C07376=1109.585,-100.826,-47.204,179.816,4.533,148.808
C07377=1109.580,-100.611,-47.213,179.815,4.537,148.809
C07378=1109.575,-100.396,-47.221,179.814,4.541,148.810
C07379=1109.571,-100.182,-47.230,179.814,4.545,148.811
C07380=1109.566,-99.966,-47.239,179.814,4.550,148.812
C07381=1109.561,-99.752,-47.247,179.814,4.555,148.813
C07382=1109.557,-99.538,-47.256,179.813,4.559,148.814
C07383=1109.553,-99.322,-47.264,179.813,4.562,148.815
C07384=1109.547,-99.073,-47.275,179.813,4.568,148.816
C07385=1109.542,-98.823,-47.285,179.813,4.573,148.817
C07386=1109.537,-98.574,-47.294,179.812,4.578,148.818
C07387=1109.532,-98.323,-47.304,179.812,4.582,148.820
C07388=1109.526,-98.074,-47.315,179.811,4.587,148.821
C07389=1109.520,-97.824,-47.325,179.811,4.593,148.822
C07390=1109.516,-97.575,-47.334,179.810,4.597,148.823
C07391=1109.511,-97.325,-47.345,179.810,4.602,148.824
C07392=1109.505,-97.075,-47.355,179.810,4.607,148.826
C07393=1109.499,-96.826,-47.365,179.810,4.612,148.827
C07394=1109.495,-96.576,-47.375,179.809,4.617,148.828
C07395=1109.489,-96.325,-47.385,179.809,4.622,148.829
C07396=1109.484,-96.076,-47.395,179.809,4.627,148.830
C07397=1109.479,-95.826,-47.406,179.808,4.631,148.832
C07398=1109.474,-95.576,-47.415,179.808,4.637,148.833
C07399=1109.468,-95.327,-47.425,179.807,4.642,148.834
C07400=1109.463,-95.077,-47.436,179.807,4.647,148.835
C07401=1109.458,-94.827,-47.446,179.806,4.651,148.836
C07402=1109.452,-94.578,-47.456,179.806,4.656,148.838
C07403=1109.447,-94.328,-47.466,179.806,4.661,148.839
C07404=1109.442,-94.078,-47.477,179.805,4.666,148.840
C07405=1109.437,-93.829,-47.487,179.805,4.671,148.841
C07406=1109.431,-93.579,-47.497,179.804,4.675,148.842
C07407=1109.426,-93.329,-47.508,179.804,4.680,148.844
C07408=1109.420,-93.079,-47.518,179.804,4.686,148.845
C07409=1109.416,-92.830,-47.527,179.803,4.690,148.846
C07410=1109.411,-92.580,-47.538,179.803,4.695,148.847
C07411=1109.405,-92.330,-47.548,179.803,4.700,148.848
C07412=1109.400,-92.080,-47.559,179.801,4.705,148.850
C07413=1109.394,-91.830,-47.569,179.801,4.710,148.851
C07414=1109.389,-91.581,-47.579,179.800,4.714,148.852
C07415=1109.384,-91.331,-47.589,179.800,4.720,148.853
C07416=1109.379,-91.081,-47.599,179.800,4.725,148.854
C07417=1109.373,-90.832,-47.610,179.799,4.729,148.856
C07418=1109.368,-90.582,-47.620,179.799,4.734,148.857
C07419=1109.363,-90.332,-47.630,179.799,4.739,148.858
C07420=1109.358,-90.082,-47.641,179.799,4.745,148.859
C07421=1109.352,-89.832,-47.651,179.797,4.749,148.861
C07422=1109.346,-89.583,-47.661,179.797,4.754,148.862
C07423=1109.342,-89.333,-47.673,179.797,4.760,148.863
C07424=1109.337,-89.084,-47.682,179.796,4.764,148.864
C07425=1109.332,-88.834,-47.693,179.796,4.769,148.865
C07426=1109.326,-88.584,-47.703,179.796,4.774,148.867
C07427=1109.321,-88.335,-47.713,179.796,4.779,148.868
C07428=1109.316,-88.084,-47.724,179.795,4.784,148.869
C07429=1109.310,-87.835,-47.734,179.794,4.789,148.870
C07430=1109.305,-87.585,-47.745,179.794,4.794,148.872
C07431=1109.300,-87.336,-47.756,179.794,4.799,148.873
C07432=1109.296,-87.120,-47.764,179.793,4.803,148.874
C07433=1109.291,-86.906,-47.773,179.793,4.808,148.875
C07434=1109.286,-86.692,-47.782,179.792,4.812,148.876
C07435=1109.282,-86.476,-47.791,179.793,4.817,148.877
C07436=1109.277,-86.262,-47.800,179.792,4.821,148.878
C07437=1109.273,-86.047,-47.810,179.792,4.825,148.879
C07438=1109.268,-85.832,-47.818,179.791,4.830,148.880
C07439=1109.263,-85.618,-47.827,179.791,4.834,148.881
C07440=1109.259,-85.368,-47.838,179.791,4.839,148.882
C07441=1109.253,-85.119,-47.849,179.791,4.844,148.883
C07442=1109.248,-84.868,-47.859,179.790,4.849,148.885
C07443=1109.242,-84.619,-47.869,179.790,4.854,148.886
C07444=1109.238,-84.369,-47.881,179.789,4.859,148.887
C07445=1109.232,-84.120,-47.891,179.789,4.864,148.888
C07446=1109.227,-83.869,-47.901,179.789,4.869,148.889
C07447=1109.221,-83.620,-47.912,179.789,4.875,148.891
C07448=1109.217,-83.370,-47.923,179.789,4.880,148.892
C07449=1109.211,-83.121,-47.933,179.788,4.884,148.893
C07450=1109.206,-82.870,-47.944,179.788,4.889,148.894
C07451=1109.201,-82.621,-47.955,179.787,4.894,148.895
C07452=1109.196,-82.371,-47.965,179.787,4.900,148.897
C07453=1109.190,-82.122,-47.975,179.787,4.905,148.898
C07454=1109.186,-81.872,-47.987,179.786,4.910,148.899
C07455=1109.180,-81.622,-47.997,179.786,4.915,148.900
C07456=1109.175,-81.372,-48.007,179.786,4.921,148.902
C07457=1109.170,-81.123,-48.018,179.786,4.926,148.903
C07458=1109.164,-80.873,-48.030,179.786,4.931,148.904
C07459=1109.158,-80.623,-48.040,179.786,4.936,148.905
C07460=1109.154,-80.374,-48.051,179.785,4.940,148.906
C07461=1109.148,-80.124,-48.061,179.785,4.945,148.907
C07462=1109.143,-79.874,-48.072,179.785,4.951,148.909
C07463=1109.138,-79.625,-48.083,179.784,4.956,148.910
C07464=1109.133,-79.375,-48.093,179.784,4.961,148.911
C07465=1109.128,-79.125,-48.105,179.784,4.966,148.912
C07466=1109.122,-78.875,-48.115,179.784,4.971,148.913
C07467=1109.117,-78.626,-48.127,179.784,4.976,148.914
C07468=1109.111,-78.376,-48.137,179.784,4.981,148.916
C07469=1109.106,-78.126,-48.148,179.783,4.987,148.917
C07470=1109.101,-77.877,-48.158,179.783,4.992,148.918
C07471=1109.096,-77.627,-48.169,179.783,4.997,148.919
C07472=1109.090,-77.377,-48.181,179.782,5.002,148.921
C07473=1109.085,-77.127,-48.191,179.782,5.008,148.922
C07474=1109.080,-76.877,-48.202,179.782,5.013,148.923
C07475=1109.075,-76.628,-48.213,179.782,5.018,148.924
C07476=1109.070,-76.378,-48.224,179.782,5.023,148.925
C07477=1109.064,-76.128,-48.235,179.782,5.028,148.926
C07478=1109.059,-75.879,-48.246,179.782,5.033,148.928
C07479=1109.054,-75.629,-48.257,179.782,5.038,148.929
C07480=1109.049,-75.380,-48.268,179.782,5.043,148.930
C07481=1109.044,-75.129,-48.278,179.782,5.048,148.931
C07482=1109.038,-74.880,-48.290,179.781,5.053,148.932
C07483=1109.033,-74.631,-48.301,179.781,5.059,148.933
C07484=1109.028,-74.380,-48.311,179.781,5.064,148.934
C07485=1109.023,-74.131,-48.322,179.781,5.069,148.936
C07486=1109.017,-73.881,-48.334,179.781,5.074,148.937
C07487=1109.012,-73.631,-48.345,179.781,5.080,148.938
C07488=1109.008,-73.417,-48.354,179.781,5.084,148.939
C07489=1109.003,-73.202,-48.364,179.781,5.089,148.940
C07490=1108.999,-72.988,-48.373,179.781,5.093,148.941
C07491=1108.994,-72.773,-48.383,179.781,5.098,148.942
C07492=1108.989,-72.559,-48.392,179.781,5.102,148.943
C07493=1108.985,-72.343,-48.402,179.781,5.106,148.944
C07494=1108.981,-72.129,-48.411,179.781,5.110,148.945
C07495=1108.976,-71.914,-48.421,179.781,5.115,148.946
C07496=1108.972,-71.665,-48.432,179.781,5.120,148.947
C07497=1108.965,-71.415,-48.443,179.781,5.125,148.948
C07498=1108.960,-71.165,-48.454,179.781,5.131,148.949
C07499=1108.956,-70.916,-48.465,179.781,5.136,148.950
C07500=1108.949,-70.666,-48.476,179.781,5.141,148.951
C07501=1108.945,-70.416,-48.488,179.781,5.146,148.952
C07502=1108.940,-70.167,-48.499,179.781,5.151,148.954
C07503=1108.935,-69.917,-48.511,179.781,5.156,148.955
C07504=1108.929,-69.667,-48.521,179.781,5.161,148.956
C07505=1108.924,-69.418,-48.532,179.781,5.166,148.957
C07506=1108.919,-69.168,-48.544,179.781,5.172,148.958
C07507=1108.914,-68.919,-48.555,179.781,5.177,148.959
C07508=1108.908,-68.668,-48.566,179.781,5.182,148.960
C07509=1108.903,-68.418,-48.578,179.782,5.187,148.961
C07510=1108.899,-68.169,-48.589,179.781,5.192,148.962
C07511=1108.892,-67.920,-48.600,179.781,5.197,148.964
C07512=1108.888,-67.670,-48.612,179.782,5.202,148.964
C07513=1108.882,-67.420,-48.624,179.782,5.207,148.966
C07514=1108.877,-67.170,-48.634,179.781,5.212,148.967
C07515=1108.871,-66.921,-48.646,179.782,5.218,148.968
C07516=1108.867,-66.671,-48.657,179.782,5.223,148.969
C07517=1108.862,-66.421,-48.668,179.782,5.228,148.970
C07518=1108.857,-66.171,-48.680,179.783,5.233,148.971
C07519=1108.851,-65.922,-48.691,179.782,5.238,148.972
C07520=1108.846,-65.673,-48.703,179.783,5.243,148.973
C07521=1108.841,-65.422,-48.713,179.783,5.248,148.974
C07522=1108.835,-65.172,-48.725,179.783,5.252,148.975
C07523=1108.831,-64.923,-48.737,179.784,5.258,148.976
C07524=1108.825,-64.674,-48.748,179.783,5.264,148.977
C07525=1108.820,-64.424,-48.759,179.784,5.268,148.978
C07526=1108.815,-64.174,-48.771,179.784,5.273,148.980
C07527=1108.810,-63.924,-48.783,179.784,5.278,148.981
C07528=1108.804,-63.674,-48.794,179.784,5.283,148.981
C07529=1108.799,-63.425,-48.805,179.784,5.288,148.983
C07530=1108.794,-63.176,-48.817,179.785,5.294,148.984
C07531=1108.789,-62.926,-48.829,179.785,5.299,148.985
C07532=1108.784,-62.676,-48.840,179.786,5.304,148.986
C07533=1108.779,-62.426,-48.852,179.786,5.309,148.987
C07534=1108.773,-62.176,-48.864,179.786,5.313,148.988
C07535=1108.767,-61.927,-48.875,179.786,5.318,148.989
C07536=1108.763,-61.678,-48.886,179.786,5.323,148.990
C07537=1108.757,-61.428,-48.898,179.787,5.329,148.991
C07538=1108.753,-61.178,-48.910,179.788,5.334,148.992
C07539=1108.747,-60.928,-48.922,179.787,5.339,148.993
C07540=1108.742,-60.678,-48.933,179.788,5.343,148.994
C07541=1108.737,-60.428,-48.945,179.788,5.348,148.995
C07542=1108.732,-60.179,-48.957,179.789,5.353,148.996
C07543=1108.727,-59.930,-48.968,179.789,5.359,148.997
C07544=1108.722,-59.715,-48.978,179.789,5.363,148.998
C07545=1108.718,-59.501,-48.988,179.789,5.367,148.999
C07546=1108.714,-59.286,-48.998,179.789,5.370,148.999
C07547=1108.709,-59.071,-49.008,179.789,5.374,149.000
C07548=1108.705,-58.857,-49.019,179.789,5.378,149.001
C07549=1108.700,-58.642,-49.029,179.788,5.382,149.002
C07550=1108.696,-58.428,-49.039,179.788,5.386,149.003
C07551=1108.691,-58.213,-49.048,179.789,5.391,149.004
C07552=1108.686,-57.964,-49.061,179.788,5.395,149.005
C07553=1108.680,-57.714,-49.073,179.788,5.400,149.006
C07554=1108.676,-57.464,-49.084,179.788,5.405,149.007
C07555=1108.670,-57.215,-49.096,179.788,5.409,149.008
C07556=1108.665,-56.965,-49.108,179.788,5.414,149.009
C07557=1108.661,-56.716,-49.120,179.787,5.419,149.010
C07558=1108.655,-56.466,-49.132,179.788,5.423,149.011
C07559=1108.650,-56.216,-49.144,179.788,5.428,149.012
C07560=1108.645,-55.966,-49.155,179.787,5.433,149.014
C07561=1108.640,-55.716,-49.167,179.787,5.437,149.015
C07562=1108.634,-55.467,-49.179,179.787,5.443,149.016
C07563=1108.629,-55.217,-49.191,179.786,5.447,149.017
C07564=1108.624,-54.967,-49.203,179.787,5.452,149.018
C07565=1108.619,-54.717,-49.214,179.787,5.457,149.019
C07566=1108.614,-54.468,-49.227,179.786,5.461,149.020
C07567=1108.609,-54.218,-49.238,179.787,5.466,149.021
C07568=1108.604,-53.968,-49.250,179.786,5.471,149.022
C07569=1108.599,-53.719,-49.263,179.786,5.475,149.023
C07570=1108.592,-53.470,-49.274,179.786,5.480,149.024
C07571=1108.587,-53.220,-49.286,179.785,5.484,149.025
C07572=1108.583,-52.971,-49.298,179.786,5.489,149.026
C07573=1108.577,-52.721,-49.310,179.786,5.494,149.027
C07574=1108.572,-52.471,-49.322,179.785,5.499,149.029
C07575=1108.567,-52.222,-49.335,179.786,5.503,149.030
C07576=1108.562,-51.972,-49.346,179.785,5.508,149.031
C07577=1108.557,-51.722,-49.358,179.785,5.513,149.032
C07578=1108.551,-51.473,-49.370,179.785,5.518,149.033
C07579=1108.546,-51.223,-49.382,179.785,5.523,149.034
C07580=1108.541,-50.972,-49.394,179.784,5.527,149.035
C07581=1108.537,-50.723,-49.406,179.785,5.532,149.036
C07582=1108.531,-50.473,-49.418,179.784,5.536,149.037
C07583=1108.526,-50.224,-49.431,179.784,5.541,149.038
C07584=1108.521,-49.974,-49.443,179.784,5.546,149.039
C07585=1108.515,-49.724,-49.455,179.784,5.550,149.040
C07586=1108.510,-49.475,-49.467,179.784,5.555,149.041
C07587=1108.505,-49.225,-49.479,179.784,5.561,149.043
C07588=1108.500,-48.976,-49.491,179.783,5.564,149.044
C07589=1108.495,-48.726,-49.503,179.783,5.570,149.045
C07590=1108.490,-48.477,-49.516,179.783,5.575,149.046
C07591=1108.484,-48.227,-49.528,179.783,5.579,149.047
C07592=1108.479,-47.977,-49.540,179.783,5.584,149.048
C07593=1108.474,-47.727,-49.552,179.782,5.588,149.049
C07594=1108.469,-47.478,-49.565,179.782,5.593,149.050
C07595=1108.463,-47.228,-49.577,179.783,5.598,149.051
C07596=1108.458,-46.979,-49.589,179.782,5.602,149.052
C07597=1108.454,-46.729,-49.600,179.782,5.607,149.053
C07598=1108.448,-46.480,-49.613,179.782,5.612,149.054
C07599=1108.443,-46.230,-49.625,179.782,5.616,149.056
C07600=1108.439,-46.016,-49.636,179.782,5.620,149.056
C07601=1108.434,-45.801,-49.646,179.781,5.624,149.057
C07602=1108.430,-45.586,-49.657,179.781,5.628,149.058
C07603=1108.426,-45.372,-49.668,179.782,5.633,149.059
C07604=1108.421,-45.157,-49.678,179.782,5.637,149.060
C07605=1108.417,-44.943,-49.689,179.781,5.641,149.061
C07606=1108.412,-44.728,-49.699,179.781,5.645,149.062
C07607=1108.408,-44.514,-49.709,179.781,5.649,149.063
C07608=1108.403,-44.265,-49.722,179.781,5.654,149.064
C07609=1108.398,-44.014,-49.734,179.780,5.658,149.065
C07610=1108.393,-43.765,-49.747,179.780,5.663,149.066
C07611=1108.387,-43.515,-49.759,179.780,5.669,149.067
C07612=1108.382,-43.266,-49.771,179.780,5.672,149.068
C07613=1108.377,-43.017,-49.784,179.780,5.678,149.069
C07614=1108.372,-42.767,-49.796,179.779,5.682,149.071
C07615=1108.366,-42.517,-49.808,179.780,5.687,149.072
C07616=1108.362,-42.267,-49.821,179.781,5.692,149.072
C07617=1108.356,-42.017,-49.833,179.781,5.697,149.073
C07618=1108.351,-41.768,-49.846,179.781,5.702,149.075
C07619=1108.346,-41.519,-49.858,179.782,5.708,149.075
C07620=1108.341,-41.269,-49.870,179.783,5.712,149.076
C07621=1108.336,-41.019,-49.883,179.783,5.717,149.077
C07622=1108.331,-40.769,-49.896,179.784,5.722,149.078
C07623=1108.326,-40.519,-49.908,179.784,5.727,149.079
C07624=1108.320,-40.270,-49.921,179.784,5.731,149.080
C07625=1108.315,-40.020,-49.934,179.785,5.737,149.081
C07626=1108.310,-39.771,-49.946,179.786,5.742,149.082
C07627=1108.304,-39.521,-49.958,179.786,5.746,149.083
C07628=1108.300,-39.271,-49.971,179.787,5.751,149.084
C07629=1108.295,-39.022,-49.984,179.787,5.756,149.085
C07630=1108.289,-38.773,-49.996,179.788,5.761,149.085
C07631=1108.284,-38.523,-50.008,179.788,5.765,149.086
C07632=1108.279,-38.273,-50.021,179.789,5.770,149.087
C07633=1108.274,-38.023,-50.034,179.789,5.775,149.088
C07634=1108.268,-37.774,-50.047,179.789,5.779,149.089
C07635=1108.263,-37.524,-50.060,179.789,5.783,149.090
C07636=1108.258,-37.275,-50.072,179.790,5.788,149.091
C07637=1108.253,-37.024,-50.084,179.790,5.793,149.092
C07638=1108.248,-36.775,-50.097,179.791,5.798,149.093
C07639=1108.243,-36.526,-50.110,179.791,5.802,149.094
C07640=1108.237,-36.276,-50.123,179.792,5.807,149.094
C07641=1108.233,-36.026,-50.136,179.792,5.811,149.095
C07642=1108.228,-35.777,-50.148,179.792,5.815,149.096
C07643=1108.223,-35.528,-50.161,179.793,5.820,149.097
C07644=1108.217,-35.278,-50.174,179.793,5.825,149.098
C07645=1108.212,-35.028,-50.187,179.794,5.830,149.099
C07646=1108.207,-34.779,-50.200,179.794,5.834,149.100
C07647=1108.202,-34.529,-50.212,179.794,5.838,149.101
C07648=1108.197,-34.279,-50.225,179.795,5.843,149.101
C07649=1108.192,-34.029,-50.237,179.795,5.847,149.102
C07650=1108.186,-33.780,-50.250,179.795,5.851,149.103
C07651=1108.181,-33.530,-50.263,179.796,5.856,149.104
C07652=1108.176,-33.280,-50.276,179.796,5.861,149.105
C07653=1108.171,-33.031,-50.288,179.797,5.865,149.106
C07654=1108.165,-32.781,-50.302,179.796,5.869,149.107
C07655=1108.161,-32.531,-50.315,179.797,5.874,149.108
C07656=1108.157,-32.317,-50.325,179.797,5.878,149.108
C07657=1108.152,-32.103,-50.337,179.798,5.881,149.109
C07658=1108.148,-31.888,-50.347,179.797,5.885,149.110
C07659=1108.143,-31.674,-50.359,179.798,5.889,149.111
C07660=1108.139,-31.460,-50.371,179.799,5.893,149.111
C07661=1108.135,-31.246,-50.381,179.799,5.897,149.112
C07662=1108.130,-31.031,-50.393,179.799,5.901,149.113
C07663=1108.126,-30.817,-50.404,179.799,5.904,149.114
C07664=1108.121,-30.567,-50.416,179.799,5.909,149.115
C07665=1108.116,-30.317,-50.430,179.799,5.913,149.116
C07666=1108.111,-30.068,-50.442,179.800,5.918,149.117
C07667=1108.105,-29.819,-50.455,179.799,5.922,149.117
C07668=1108.100,-29.568,-50.468,179.800,5.927,149.118
C07669=1108.095,-29.319,-50.481,179.800,5.930,149.119
C07670=1108.090,-29.070,-50.494,179.800,5.935,149.120
C07671=1108.085,-28.820,-50.508,179.801,5.940,149.121
C07672=1108.080,-28.571,-50.521,179.801,5.944,149.122
C07673=1108.075,-28.320,-50.533,179.801,5.949,149.123
C07674=1108.069,-28.071,-50.547,179.801,5.953,149.124
C07675=1108.064,-27.822,-50.559,179.801,5.958,149.125
C07676=1108.059,-27.571,-50.573,179.801,5.962,149.126
C07677=1108.054,-27.323,-50.586,179.801,5.966,149.127
C07678=1108.049,-27.073,-50.599,179.802,5.971,149.128
C07679=1108.044,-26.823,-50.612,179.801,5.975,149.129
C07680=1108.039,-26.574,-50.625,179.802,5.980,149.130
C07681=1108.034,-26.324,-50.638,179.801,5.984,149.131
C07682=1108.029,-26.075,-50.652,179.801,5.989,149.132
C07683=1108.024,-25.825,-50.665,179.801,5.993,149.133
C07684=1108.018,-25.575,-50.678,179.801,5.998,149.134
C07685=1108.013,-25.326,-50.691,179.802,6.003,149.135
C07686=1108.008,-25.076,-50.705,179.802,6.008,149.136
C07687=1108.003,-24.827,-50.717,179.803,6.012,149.137
C07688=1107.999,-24.577,-50.730,179.803,6.017,149.137
C07689=1107.993,-24.327,-50.744,179.804,6.022,149.138
C07690=1107.988,-24.077,-50.757,179.803,6.026,149.139
C07691=1107.983,-23.828,-50.770,179.803,6.031,149.140
C07692=1107.978,-23.578,-50.783,179.804,6.036,149.141
C07693=1107.973,-23.329,-50.797,179.804,6.040,149.142
C07694=1107.967,-23.080,-50.810,179.805,6.045,149.143
C07695=1107.962,-22.829,-50.824,179.805,6.050,149.144
C07696=1107.957,-22.580,-50.837,179.806,6.055,149.145
C07697=1107.952,-22.330,-50.850,179.806,6.059,149.146
C07698=1107.947,-22.081,-50.863,179.807,6.064,149.147
C07699=1107.942,-21.831,-50.877,179.807,6.069,149.148
C07700=1107.937,-21.582,-50.890,179.807,6.073,149.148
C07701=1107.932,-21.331,-50.903,179.808,6.077,149.149
C07702=1107.927,-21.083,-50.917,179.808,6.082,149.150
C07703=1107.921,-20.832,-50.930,179.809,6.087,149.151
C07704=1107.916,-20.583,-50.944,179.809,6.092,149.152
C07705=1107.911,-20.333,-50.957,179.810,6.096,149.153
C07706=1107.906,-20.084,-50.970,179.810,6.101,149.154
C07707=1107.901,-19.834,-50.984,179.811,6.106,149.155
C07708=1107.895,-19.585,-50.997,179.810,6.110,149.156
C07709=1107.891,-19.335,-51.011,179.811,6.114,149.157
C07710=1107.885,-19.086,-51.024,179.811,6.119,149.157
C07711=1107.880,-18.836,-51.038,179.812,6.124,149.158
C07712=1107.876,-18.622,-51.049,179.812,6.128,149.159
C07713=1107.872,-18.408,-51.061,179.813,6.132,149.160
C07714=1107.867,-18.193,-51.072,179.813,6.136,149.161
C07715=1107.863,-17.979,-51.085,179.813,6.140,149.162
C07716=1107.859,-17.764,-51.096,179.814,6.144,149.162
C07717=1107.855,-17.551,-51.108,179.814,6.148,149.163
C07718=1107.850,-17.336,-51.119,179.814,6.151,149.164
C07719=1107.846,-17.122,-51.131,179.815,6.156,149.164
C07720=1107.840,-16.872,-51.145,179.816,6.160,149.165
C07721=1107.836,-16.623,-51.158,179.816,6.164,149.166
C07722=1107.831,-16.373,-51.172,179.816,6.169,149.167
C07723=1107.825,-16.123,-51.186,179.817,6.174,149.168
C07724=1107.820,-15.874,-51.199,179.817,6.179,149.169
C07725=1107.815,-15.624,-51.213,179.818,6.183,149.170
C07726=1107.810,-15.375,-51.226,179.818,6.188,149.171
C07727=1107.805,-15.125,-51.239,179.819,6.192,149.171
C07728=1107.800,-14.875,-51.254,179.819,6.197,149.172
C07729=1107.795,-14.626,-51.268,179.819,6.201,149.173
C07730=1107.790,-14.376,-51.281,179.820,6.206,149.174
C07731=1107.785,-14.127,-51.295,179.820,6.210,149.175
C07732=1107.780,-13.877,-51.309,179.821,6.215,149.176
C07733=1107.774,-13.627,-51.322,179.822,6.219,149.177
C07734=1107.770,-13.378,-51.336,179.822,6.224,149.177
C07735=1107.765,-13.129,-51.350,179.823,6.229,149.178
C07736=1107.759,-12.878,-51.364,179.823,6.233,149.179
C07737=1107.754,-12.629,-51.377,179.823,6.238,149.180
C07738=1107.750,-12.380,-51.391,179.824,6.242,149.181
C07739=1107.745,-12.130,-51.405,179.825,6.247,149.182
C07740=1107.739,-11.881,-51.419,179.825,6.251,149.183
C07741=1107.734,-11.631,-51.433,179.826,6.256,149.184
C07742=1107.730,-11.382,-51.447,179.826,6.261,149.184
C07743=1107.724,-11.133,-51.460,179.827,6.264,149.185
C07744=1107.719,-10.882,-51.474,179.827,6.269,149.186
C07745=1107.714,-10.632,-51.488,179.828,6.274,149.187
C07746=1107.708,-10.383,-51.502,179.828,6.278,149.188
C07747=1107.704,-10.134,-51.516,179.829,6.283,149.189
C07748=1107.699,-9.884,-51.530,179.830,6.288,149.189
C07749=1107.693,-9.635,-51.543,179.830,6.292,149.190
C07750=1107.688,-9.385,-51.558,179.831,6.297,149.191
C07751=1107.683,-9.135,-51.572,179.831,6.301,149.192
C07752=1107.679,-8.886,-51.586,179.832,6.305,149.193
C07753=1107.673,-8.637,-51.600,179.832,6.310,149.194
C07754=1107.669,-8.387,-51.614,179.833,6.315,149.194
C07755=1107.663,-8.137,-51.627,179.833,6.319,149.195
C07756=1107.658,-7.888,-51.641,179.834,6.324,149.196
C07757=1107.653,-7.638,-51.656,179.835,6.328,149.197
C07758=1107.648,-7.388,-51.670,179.835,6.333,149.198
C07759=1107.643,-7.139,-51.684,179.835,6.337,149.199
C07760=1107.637,-6.890,-51.698,179.836,6.341,149.199
C07761=1107.633,-6.640,-51.712,179.836,6.346,149.200
C07762=1107.628,-6.391,-51.726,179.837,6.351,149.201
C07763=1107.623,-6.141,-51.740,179.838,6.355,149.202
C07764=1107.618,-5.892,-51.754,179.838,6.360,149.203
C07765=1107.613,-5.642,-51.768,179.839,6.365,149.204
C07766=1107.608,-5.392,-51.783,179.840,6.369,149.205
C07767=1107.603,-5.143,-51.797,179.840,6.373,149.205
C07768=1107.598,-4.929,-51.809,179.840,6.378,149.206
C07769=1107.594,-4.715,-51.821,179.841,6.381,149.207
C07770=1107.590,-4.500,-51.833,179.841,6.385,149.207
C07771=1107.586,-4.286,-51.845,179.842,6.389,149.208
C07772=1107.581,-4.072,-51.857,179.843,6.393,149.209
C07773=1107.576,-3.857,-51.870,179.843,6.396,149.209
C07774=1107.572,-3.643,-51.882,179.844,6.401,149.210
C07775=1107.567,-3.429,-51.894,179.844,6.404,149.211
C07776=1107.563,-3.180,-51.909,179.844,6.409,149.212
C07777=1107.558,-2.930,-51.923,179.845,6.413,149.213
C07778=1107.553,-2.680,-51.937,179.846,6.418,149.213
C07779=1107.548,-2.431,-51.952,179.846,6.423,149.214
C07780=1107.543,-2.181,-51.966,179.847,6.427,149.215
C07781=1107.537,-1.932,-51.980,179.848,6.432,149.216
C07782=1107.532,-1.682,-51.994,179.848,6.436,149.217
C07783=1107.527,-1.433,-52.008,179.848,6.440,149.218
C07784=1107.522,-1.183,-52.023,179.849,6.445,149.218
C07785=1107.517,-0.933,-52.037,179.850,6.450,149.219
C07786=1107.513,-0.684,-52.052,179.850,6.454,149.220
C07787=1107.507,-0.435,-52.066,179.851,6.459,149.221
C07788=1107.502,-0.185,-52.080,179.852,6.463,149.222
C07789=1107.497,0.064,-52.094,179.853,6.468,149.223
C07790=1107.492,0.314,-52.109,179.854,6.472,149.223
C07791=1107.487,0.563,-52.124,179.854,6.477,149.224
C07792=1107.482,0.813,-52.139,179.855,6.482,149.225
C07793=1107.477,1.063,-52.153,179.855,6.486,149.226
C07794=1107.472,1.313,-52.167,179.856,6.490,149.227
C07795=1107.467,1.562,-52.181,179.856,6.495,149.227
C07796=1107.462,1.811,-52.196,179.857,6.499,149.228
C07797=1107.457,2.060,-52.210,179.857,6.504,149.229
C07798=1107.452,2.310,-52.225,179.858,6.508,149.230
C07799=1107.447,2.560,-52.240,179.859,6.513,149.231
C07800=1107.442,2.809,-52.254,179.859,6.518,149.232
C07801=1107.437,3.059,-52.269,179.860,6.522,149.232
C07802=1107.432,3.309,-52.283,179.861,6.527,149.233
C07803=1107.427,3.558,-52.298,179.861,6.532,149.234
C07804=1107.422,3.807,-52.312,179.862,6.536,149.235
C07805=1107.416,4.057,-52.327,179.863,6.541,149.236
C07806=1107.412,4.307,-52.342,179.863,6.545,149.237
C07807=1107.407,4.556,-52.356,179.864,6.550,149.237
C07808=1107.402,4.806,-52.371,179.864,6.555,149.238
C07809=1107.396,5.055,-52.386,179.865,6.559,149.239
C07810=1107.391,5.305,-52.401,179.866,6.564,149.240
C07811=1107.387,5.554,-52.416,179.867,6.569,149.241
C07812=1107.382,5.804,-52.430,179.867,6.573,149.242
C07813=1107.376,6.053,-52.444,179.868,6.578,149.242
C07814=1107.371,6.302,-52.459,179.869,6.582,149.243
C07815=1107.366,6.552,-52.474,179.869,6.587,149.244
C07816=1107.361,6.801,-52.489,179.870,6.592,149.245
C07817=1107.356,7.051,-52.503,179.870,6.596,149.246
C07818=1107.351,7.300,-52.518,179.871,6.601,149.247
C07819=1107.346,7.550,-52.533,179.872,6.605,149.247
C07820=1107.341,7.799,-52.548,179.872,6.610,149.248
C07821=1107.336,8.049,-52.563,179.873,6.615,149.249
C07822=1107.331,8.298,-52.578,179.874,6.619,149.250
C07823=1107.327,8.549,-52.592,179.874,6.624,149.251
C07824=1107.322,8.762,-52.606,179.874,6.628,149.252
C07825=1107.318,8.977,-52.618,179.875,6.631,149.252
C07826=1107.313,9.191,-52.630,179.875,6.635,149.253
C07827=1107.309,9.405,-52.644,179.876,6.640,149.254
C07828=1107.305,9.619,-52.656,179.876,6.643,149.255
C07829=1107.300,9.833,-52.669,179.876,6.647,149.255
C07830=1107.296,10.047,-52.681,179.877,6.651,149.256
C07831=1107.292,10.261,-52.695,179.877,6.654,149.257
C07832=1107.287,10.511,-52.709,179.877,6.659,149.258
C07833=1107.282,10.760,-52.724,179.878,6.663,149.259
C07834=1107.277,11.010,-52.740,179.879,6.668,149.259
C07835=1107.272,11.259,-52.754,179.879,6.672,149.260
C07836=1107.267,11.509,-52.769,179.879,6.677,149.261
C07837=1107.261,11.759,-52.784,179.880,6.682,149.262
C07838=1107.257,12.008,-52.799,179.880,6.686,149.263
C07839=1107.251,12.257,-52.815,179.881,6.690,149.264
C07840=1107.246,12.507,-52.829,179.881,6.694,149.265
C07841=1107.242,12.756,-52.844,179.882,6.699,149.265
C07842=1107.236,13.005,-52.860,179.882,6.704,149.266
C07843=1107.231,13.255,-52.874,179.882,6.708,149.267
C07844=1107.227,13.505,-52.890,179.883,6.712,149.268
C07845=1107.222,13.754,-52.905,179.884,6.717,149.269
C07846=1107.216,14.004,-52.920,179.884,6.721,149.270
C07847=1107.212,14.253,-52.935,179.884,6.725,149.271
C07848=1107.207,14.502,-52.950,179.885,6.730,149.271
C07849=1107.202,14.752,-52.965,179.886,6.734,149.272
C07850=1107.197,15.002,-52.980,179.886,6.739,149.273
C07851=1107.191,15.251,-52.995,179.886,6.743,149.274
C07852=1107.187,15.501,-53.011,179.887,6.747,149.274
C07853=1107.182,15.750,-53.026,179.888,6.752,149.275
C07854=1107.177,16.000,-53.040,179.889,6.757,149.276
C07855=1107.171,16.249,-53.056,179.889,6.760,149.277
C07856=1107.167,16.498,-53.071,179.890,6.765,149.278
C07857=1107.161,16.748,-53.087,179.890,6.770,149.279
C07858=1107.157,16.998,-53.102,179.891,6.774,149.279
C07859=1107.152,17.248,-53.117,179.891,6.778,149.280
C07860=1107.146,17.497,-53.132,179.892,6.783,149.281
C07861=1107.142,17.746,-53.147,179.893,6.787,149.282
C07862=1107.136,17.995,-53.163,179.893,6.791,149.283
C07863=1107.132,18.245,-53.178,179.893,6.796,149.284
C07864=1107.127,18.495,-53.194,179.894,6.800,149.284
C07865=1107.122,18.744,-53.209,179.895,6.805,149.285
C07866=1107.116,18.994,-53.224,179.895,6.808,149.286
C07867=1107.112,19.243,-53.239,179.896,6.813,149.287
C07868=1107.106,19.492,-53.254,179.896,6.817,149.288
C07869=1107.102,19.742,-53.270,179.897,6.822,149.288
C07870=1107.097,19.991,-53.285,179.897,6.826,149.289
C07871=1107.092,20.241,-53.301,179.898,6.830,149.290
C07872=1107.086,20.490,-53.316,179.899,6.835,149.291
C07873=1107.082,20.740,-53.332,179.900,6.839,149.291
C07874=1107.077,20.989,-53.347,179.900,6.843,149.292
C07875=1107.072,21.239,-53.362,179.901,6.847,149.293
C07876=1107.067,21.488,-53.378,179.902,6.852,149.294
C07877=1107.061,21.737,-53.394,179.902,6.855,149.294
C07878=1107.057,21.987,-53.409,179.903,6.860,149.295
C07879=1107.052,22.237,-53.425,179.904,6.865,149.296
C07880=1107.048,22.451,-53.438,179.904,6.868,149.297
C07881=1107.044,22.664,-53.451,179.904,6.872,149.297
C07882=1107.039,22.878,-53.465,179.905,6.875,149.298
C07883=1107.035,23.093,-53.478,179.906,6.879,149.299
C07884=1107.030,23.307,-53.490,179.906,6.883,149.299
C07885=1107.026,23.521,-53.504,179.907,6.886,149.300
C07886=1107.022,23.735,-53.518,179.907,6.890,149.300
C07887=1107.018,23.949,-53.531,179.908,6.893,149.301
C07888=1107.013,24.199,-53.547,179.909,6.898,149.302
C07889=1107.008,24.448,-53.562,179.909,6.902,149.303
C07890=1107.003,24.697,-53.577,179.910,6.907,149.303
C07891=1106.998,24.946,-53.593,179.910,6.911,149.304
C07892=1106.993,25.196,-53.609,179.911,6.915,149.305
C07893=1106.988,25.446,-53.625,179.912,6.919,149.306
C07894=1106.983,25.695,-53.640,179.912,6.923,149.306
C07895=1106.978,25.945,-53.656,179.913,6.928,149.307
C07896=1106.973,26.194,-53.672,179.914,6.932,149.308
C07897=1106.967,26.444,-53.687,179.915,6.937,149.309
C07898=1106.963,26.693,-53.704,179.916,6.940,149.309
C07899=1106.958,26.942,-53.719,179.917,6.944,149.310
C07900=1106.953,27.192,-53.734,179.917,6.949,149.311
C07901=1106.948,27.442,-53.750,179.918,6.953,149.311
C07902=1106.943,27.691,-53.766,179.919,6.957,149.312
C07903=1106.938,27.940,-53.782,179.920,6.961,149.313
C07904=1106.934,28.190,-53.798,179.920,6.966,149.314
C07905=1106.928,28.439,-53.813,179.921,6.969,149.314
C07906=1106.923,28.688,-53.829,179.922,6.974,149.315
C07907=1106.918,28.938,-53.845,179.922,6.978,149.316
C07908=1106.913,29.187,-53.861,179.923,6.983,149.317
C07909=1106.909,29.437,-53.876,179.924,6.986,149.317
C07910=1106.904,29.686,-53.892,179.925,6.991,149.318
C07911=1106.898,29.935,-53.908,179.926,6.995,149.319
C07912=1106.894,30.185,-53.924,179.926,6.999,149.319
C07913=1106.888,30.435,-53.940,179.927,7.003,149.320
C07914=1106.884,30.684,-53.956,179.928,7.007,149.321
C07915=1106.878,30.934,-53.972,179.929,7.012,149.321
C07916=1106.873,31.183,-53.988,179.929,7.016,149.322
C07917=1106.869,31.433,-54.004,179.930,7.020,149.323
C07918=1106.864,31.682,-54.019,179.931,7.024,149.324
C07919=1106.859,31.932,-54.035,179.932,7.028,149.324
C07920=1106.854,32.181,-54.052,179.933,7.032,149.325
C07921=1106.849,32.430,-54.067,179.934,7.036,149.326
C07922=1106.844,32.679,-54.084,179.935,7.041,149.326
C07923=1106.839,32.929,-54.099,179.935,7.045,149.327
C07924=1106.834,33.179,-54.115,179.936,7.049,149.328
C07925=1106.829,33.428,-54.132,179.937,7.053,149.328
C07926=1106.824,33.678,-54.148,179.938,7.058,149.329
C07927=1106.819,33.927,-54.164,179.938,7.061,149.330
C07928=1106.814,34.177,-54.180,179.940,7.065,149.330
C07929=1106.809,34.425,-54.196,179.941,7.070,149.331
C07930=1106.804,34.675,-54.212,179.941,7.073,149.332
C07931=1106.799,34.924,-54.228,179.942,7.077,149.332
C07932=1106.794,35.174,-54.244,179.943,7.082,149.333
C07933=1106.789,35.423,-54.261,179.944,7.086,149.334
C07934=1106.784,35.673,-54.276,179.944,7.090,149.334
C07935=1106.780,35.922,-54.293,179.945,7.094,149.335
C07936=1106.775,36.136,-54.307,179.946,7.097,149.336
C07937=1106.770,36.350,-54.320,179.947,7.101,149.336
C07938=1106.766,36.564,-54.334,179.948,7.105,149.337
C07939=1106.762,36.778,-54.348,179.949,7.108,149.337
C07940=1106.758,36.992,-54.362,179.949,7.112,149.338
C07941=1106.754,37.206,-54.376,179.950,7.115,149.338
C07942=1106.750,37.420,-54.390,179.950,7.119,149.339
C07943=1106.745,37.633,-54.404,179.952,7.122,149.340
C07944=1106.740,37.884,-54.420,179.952,7.126,149.340
C07945=1106.735,38.132,-54.436,179.953,7.130,149.341
C07946=1106.730,38.382,-54.452,179.955,7.135,149.341
C07947=1106.726,38.632,-54.469,179.956,7.139,149.342
C07948=1106.721,38.881,-54.485,179.956,7.142,149.343
C07949=1106.716,39.131,-54.501,179.957,7.147,149.343
C07950=1106.711,39.380,-54.517,179.958,7.151,149.344
C07951=1106.706,39.629,-54.534,179.959,7.155,149.345
C07952=1106.700,39.879,-54.550,179.960,7.159,149.345
C07953=1106.696,40.128,-54.567,179.961,7.163,149.346
C07954=1106.691,40.377,-54.583,179.962,7.167,149.347
C07955=1106.686,40.627,-54.599,179.962,7.171,149.347
C07956=1106.681,40.877,-54.616,179.963,7.175,149.348
C07957=1106.676,41.125,-54.632,179.964,7.180,149.349
C07958=1106.672,41.375,-54.649,179.966,7.184,149.349
C07959=1106.666,41.625,-54.665,179.966,7.187,149.350
C07960=1106.661,41.874,-54.682,179.968,7.191,149.350
C07961=1106.656,42.123,-54.698,179.969,7.196,149.351
C07962=1106.652,42.372,-54.715,179.969,7.199,149.352
C07963=1106.647,42.622,-54.731,179.970,7.203,149.352
C07964=1106.641,42.872,-54.748,179.971,7.208,149.353
C07965=1106.637,43.121,-54.764,179.972,7.212,149.354
C07966=1106.632,43.371,-54.781,179.973,7.216,149.354
C07967=1106.627,43.619,-54.797,179.974,7.219,149.355
C07968=1106.622,43.869,-54.813,179.975,7.224,149.355
C07969=1106.616,44.119,-54.830,179.976,7.228,149.356
C07970=1106.612,44.368,-54.847,179.977,7.232,149.357
C07971=1106.607,44.617,-54.863,179.978,7.236,149.357
C07972=1106.602,44.866,-54.880,179.979,7.240,149.358
C07973=1106.597,45.116,-54.897,179.981,7.244,149.359
C07974=1106.593,45.366,-54.914,179.981,7.248,149.359
C07975=1106.588,45.614,-54.930,179.982,7.252,149.360
C07976=1106.582,45.865,-54.946,179.983,7.256,149.360
C07977=1106.578,46.114,-54.963,179.985,7.260,149.361
C07978=1106.573,46.363,-54.979,179.985,7.264,149.362
C07979=1106.568,46.612,-54.996,179.986,7.268,149.362
C07980=1106.563,46.862,-55.013,179.987,7.272,149.363
C07981=1106.558,47.111,-55.030,179.989,7.277,149.364
C07982=1106.553,47.361,-55.046,179.989,7.280,149.364
C07983=1106.548,47.610,-55.064,179.991,7.284,149.365
C07984=1106.544,47.860,-55.080,179.992,7.288,149.365
C07985=1106.539,48.109,-55.097,179.993,7.293,149.366
C07986=1106.533,48.358,-55.114,179.994,7.296,149.366
C07987=1106.529,48.608,-55.131,179.995,7.300,149.367
C07988=1106.524,48.857,-55.147,179.996,7.304,149.368
C07989=1106.519,49.106,-55.164,179.997,7.308,149.368
C07990=1106.514,49.356,-55.181,179.998,7.312,149.369
C07991=1106.509,49.606,-55.198,179.999,7.316,149.369
C07992=1106.505,49.819,-55.212,180.000,7.319,149.370
C07993=1106.501,50.033,-55.227,-179.999,7.323,149.370
C07994=1106.497,50.247,-55.241,-179.998,7.327,149.371
C07995=1106.492,50.461,-55.256,-179.997,7.330,149.371
C07996=1106.488,50.675,-55.271,-179.996,7.333,149.372
C07997=1106.484,50.888,-55.285,-179.996,7.336,149.372
C07998=1106.480,51.103,-55.299,-179.994,7.340,149.373
C07999=1106.475,51.317,-55.314,-179.993,7.343,149.373
C08000=1106.470,51.565,-55.331,-179.992,7.348,149.374
C08001=1106.466,51.814,-55.348,-179.992,7.351,149.375
C08002=1106.461,52.064,-55.365,-179.990,7.355,149.375
C08003=1106.456,52.314,-55.381,-179.989,7.359,149.376
C08004=1106.451,52.563,-55.399,-179.988,7.363,149.376
C08005=1106.446,52.812,-55.415,-179.987,7.367,149.377
C08006=1106.441,53.061,-55.433,-179.986,7.371,149.377
C08007=1106.436,53.311,-55.450,-179.984,7.375,149.378
C08008=1106.431,53.561,-55.467,-179.983,7.379,149.379
C08009=1106.427,53.810,-55.484,-179.982,7.384,149.379
C08010=1106.421,54.059,-55.501,-179.981,7.387,149.380
C08011=1106.417,54.308,-55.518,-179.980,7.391,149.380
C08012=1106.412,54.558,-55.535,-179.979,7.395,149.381
C08013=1106.406,54.808,-55.552,-179.978,7.399,149.381
C08014=1106.402,55.057,-55.569,-179.977,7.403,149.382
C08015=1106.396,55.306,-55.587,-179.976,7.407,149.382
C08016=1106.392,55.555,-55.603,-179.975,7.411,149.383
C08017=1106.387,55.805,-55.621,-179.973,7.415,149.384
C08018=1106.382,56.054,-55.638,-179.972,7.419,149.384
C08019=1106.377,56.304,-55.655,-179.971,7.422,149.385
C08020=1106.372,56.553,-55.673,-179.970,7.427,149.385
C08021=1106.368,56.802,-55.690,-179.969,7.431,149.386
C08022=1106.362,57.051,-55.707,-179.967,7.435,149.386
C08023=1106.358,57.301,-55.724,-179.967,7.438,149.387
C08024=1106.353,57.550,-55.742,-179.965,7.442,149.387
C08025=1106.347,57.800,-55.759,-179.964,7.446,149.388
C08026=1106.343,58.049,-55.776,-179.962,7.450,149.389
C08027=1106.338,58.298,-55.793,-179.961,7.455,149.389
C08028=1106.334,58.548,-55.810,-179.960,7.458,149.390
C08029=1106.329,58.797,-55.828,-179.959,7.462,149.390
C08030=1106.323,59.047,-55.845,-179.958,7.466,149.391
C08031=1106.319,59.295,-55.862,-179.957,7.470,149.391
C08032=1106.313,59.545,-55.880,-179.955,7.474,149.392
C08033=1106.309,59.794,-55.898,-179.955,7.478,149.392
C08034=1106.304,60.043,-55.914,-179.953,7.482,149.393
C08035=1106.299,60.293,-55.932,-179.952,7.486,149.394
C08036=1106.294,60.542,-55.950,-179.950,7.490,149.394
C08037=1106.289,60.792,-55.967,-179.949,7.494,149.395
C08038=1106.285,61.041,-55.984,-179.948,7.497,149.395
C08039=1106.280,61.290,-56.002,-179.947,7.501,149.396
C08040=1106.274,61.540,-56.019,-179.946,7.505,149.396
C08041=1106.270,61.789,-56.037,-179.945,7.510,149.397
C08042=1106.265,62.039,-56.054,-179.943,7.514,149.397
C08043=1106.260,62.288,-56.072,-179.942,7.518,149.398
C08044=1106.255,62.537,-56.090,-179.941,7.521,149.398
C08045=1106.251,62.787,-56.107,-179.940,7.525,149.399
C08046=1106.246,63.036,-56.125,-179.938,7.529,149.399
C08047=1106.241,63.286,-56.142,-179.937,7.533,149.400
C08048=1106.237,63.499,-56.157,-179.936,7.537,149.401
C08049=1106.232,63.713,-56.172,-179.935,7.540,149.401
C08050=1106.227,63.927,-56.187,-179.934,7.544,149.401
C08051=1106.224,64.140,-56.202,-179.933,7.547,149.402
C08052=1106.220,64.354,-56.218,-179.932,7.550,149.402
C08053=1106.216,64.567,-56.233,-179.930,7.554,149.403
C08054=1106.211,64.781,-56.248,-179.929,7.557,149.403
C08055=1106.207,64.995,-56.262,-179.928,7.560,149.404
C08056=1106.202,65.244,-56.280,-179.927,7.564,149.404
C08057=1106.197,65.494,-56.298,-179.926,7.568,149.405
C08058=1106.193,65.743,-56.316,-179.924,7.572,149.405
C08059=1106.187,65.993,-56.333,-179.924,7.576,149.406
C08060=1106.182,66.242,-56.351,-179.922,7.579,149.406
C08061=1106.179,66.491,-56.369,-179.921,7.584,149.407
C08062=1106.174,66.740,-56.387,-179.919,7.588,149.407
C08063=1106.169,66.990,-56.404,-179.918,7.592,149.408
C08064=1106.164,67.239,-56.422,-179.917,7.596,149.408
C08065=1106.159,67.489,-56.440,-179.916,7.599,149.409
C08066=1106.154,67.738,-56.458,-179.915,7.603,149.409
C08067=1106.149,67.987,-56.476,-179.913,7.607,149.410
C08068=1106.144,68.237,-56.494,-179.912,7.611,149.410
C08069=1106.139,68.486,-56.512,-179.910,7.615,149.411
C08070=1106.134,68.735,-56.530,-179.909,7.619,149.411
C08071=1106.130,68.984,-56.547,-179.907,7.623,149.412
C08072=1106.125,69.233,-56.565,-179.907,7.627,149.413
C08073=1106.120,69.482,-56.583,-179.905,7.631,149.413
C08074=1106.116,69.732,-56.601,-179.904,7.634,149.413
C08075=1106.110,69.982,-56.618,-179.903,7.639,149.414
C08076=1106.106,70.231,-56.636,-179.901,7.643,149.414
C08077=1106.101,70.480,-56.654,-179.899,7.647,149.415
C08078=1106.096,70.729,-56.672,-179.898,7.651,149.416
C08079=1106.091,70.979,-56.690,-179.897,7.655,149.416
C08080=1106.086,71.228,-56.708,-179.896,7.658,149.416
C08081=1106.082,71.478,-56.727,-179.895,7.662,149.417
C08082=1106.077,71.727,-56.745,-179.893,7.666,149.418
C08083=1106.072,71.976,-56.763,-179.892,7.670,149.418
C08084=1106.067,72.225,-56.781,-179.890,7.674,149.419
C08085=1106.062,72.474,-56.799,-179.889,7.678,149.419
C08086=1106.057,72.724,-56.817,-179.887,7.682,149.419
C08087=1106.052,72.973,-56.835,-179.886,7.686,149.420
C08088=1106.047,73.223,-56.854,-179.885,7.689,149.421
C08089=1106.042,73.472,-56.872,-179.884,7.693,149.421
C08090=1106.037,73.721,-56.890,-179.883,7.698,149.422
C08091=1106.032,73.970,-56.907,-179.881,7.702,149.422
C08092=1106.027,74.220,-56.925,-179.879,7.705,149.423
C08093=1106.023,74.470,-56.944,-179.878,7.710,149.423
C08094=1106.019,74.718,-56.963,-179.877,7.714,149.424
C08095=1106.014,74.967,-56.980,-179.875,7.718,149.424
C08096=1106.009,75.216,-56.998,-179.874,7.721,149.424
C08097=1106.004,75.466,-57.016,-179.872,7.726,149.425
C08098=1105.999,75.716,-57.035,-179.871,7.729,149.426
C08099=1105.994,75.965,-57.053,-179.870,7.733,149.426
C08100=1105.989,76.214,-57.071,-179.869,7.737,149.427
C08101=1105.984,76.463,-57.090,-179.867,7.741,149.427
C08102=1105.980,76.713,-57.108,-179.866,7.745,149.428
C08103=1105.975,76.962,-57.126,-179.864,7.749,149.428
C08104=1105.971,77.175,-57.142,-179.864,7.752,149.429
C08105=1105.967,77.389,-57.158,-179.863,7.755,149.429
C08106=1105.962,77.603,-57.174,-179.862,7.758,149.429
C08107=1105.958,77.816,-57.190,-179.861,7.762,149.430
C08108=1105.954,78.031,-57.205,-179.860,7.765,149.430
C08109=1105.949,78.244,-57.221,-179.859,7.768,149.431
C08110=1105.946,78.458,-57.237,-179.858,7.771,149.431
C08111=1105.941,78.672,-57.253,-179.857,7.774,149.432
C08112=1105.937,78.920,-57.271,-179.857,7.778,149.433
C08113=1105.932,79.169,-57.289,-179.855,7.782,149.433
C08114=1105.927,79.419,-57.308,-179.855,7.785,149.434
C08115=1105.922,79.668,-57.326,-179.853,7.789,149.434
C08116=1105.917,79.917,-57.345,-179.853,7.793,149.435
C08117=1105.913,80.167,-57.363,-179.851,7.797,149.435
C08118=1105.908,80.416,-57.381,-179.851,7.800,149.436
C08119=1105.903,80.665,-57.401,-179.849,7.804,149.436
C08120=1105.898,80.915,-57.419,-179.848,7.807,149.437
C08121=1105.893,81.164,-57.437,-179.847,7.812,149.437
C08122=1105.889,81.413,-57.456,-179.846,7.815,149.438
C08123=1105.884,81.663,-57.474,-179.845,7.819,149.439
C08124=1105.879,81.912,-57.493,-179.844,7.822,149.439
C08125=1105.874,82.161,-57.511,-179.843,7.826,149.440
C08126=1105.869,82.411,-57.530,-179.842,7.830,149.440
C08127=1105.865,82.659,-57.549,-179.841,7.834,149.441
C08128=1105.860,82.909,-57.567,-179.839,7.838,149.441
C08129=1105.855,83.158,-57.586,-179.839,7.841,149.442
C08130=1105.850,83.407,-57.604,-179.837,7.845,149.442
C08131=1105.845,83.656,-57.623,-179.837,7.849,149.443
C08132=1105.840,83.906,-57.642,-179.835,7.853,149.443
C08133=1105.835,84.155,-57.660,-179.834,7.857,149.444
C08134=1105.831,84.404,-57.679,-179.833,7.860,149.444
C08135=1105.826,84.654,-57.698,-179.832,7.864,149.445
C08136=1105.821,84.903,-57.716,-179.831,7.867,149.446
C08137=1105.817,85.152,-57.735,-179.829,7.871,149.446
C08138=1105.811,85.401,-57.754,-179.828,7.875,149.447
C08139=1105.807,85.650,-57.773,-179.827,7.879,149.447
C08140=1105.802,85.900,-57.792,-179.826,7.883,149.448
C08141=1105.797,86.149,-57.810,-179.825,7.886,149.448
C08142=1105.792,86.399,-57.829,-179.824,7.890,149.449
C08143=1105.788,86.647,-57.848,-179.823,7.894,149.449
C08144=1105.783,86.897,-57.866,-179.822,7.897,149.450
C08145=1105.778,87.146,-57.886,-179.820,7.902,149.450
C08146=1105.773,87.395,-57.904,-179.819,7.905,149.451
C08147=1105.768,87.645,-57.923,-179.818,7.909,149.451
C08148=1105.764,87.893,-57.942,-179.817,7.913,149.452
C08149=1105.759,88.144,-57.961,-179.816,7.916,149.452
C08150=1105.754,88.392,-57.980,-179.815,7.920,149.453
C08151=1105.749,88.642,-57.999,-179.813,7.924,149.453
C08152=1105.744,88.891,-58.017,-179.812,7.927,149.454
C08153=1105.739,89.140,-58.036,-179.811,7.931,149.454
C08154=1105.735,89.389,-58.056,-179.809,7.935,149.455
C08155=1105.729,89.639,-58.074,-179.808,7.939,149.455
C08156=1105.725,89.888,-58.093,-179.807,7.943,149.456
C08157=1105.720,90.137,-58.112,-179.806,7.947,149.456
C08158=1105.716,90.386,-58.132,-179.804,7.951,149.457
C08159=1105.710,90.635,-58.150,-179.804,7.954,149.457
C08160=1105.707,90.849,-58.167,-179.803,7.957,149.458
C08161=1105.702,91.062,-58.183,-179.801,7.961,149.458
C08162=1105.699,91.276,-58.199,-179.800,7.964,149.459
C08163=1105.695,91.490,-58.216,-179.799,7.967,149.459
C08164=1105.690,91.704,-58.232,-179.798,7.970,149.459
C08165=1105.686,91.917,-58.249,-179.797,7.973,149.460
C08166=1105.682,92.130,-58.264,-179.796,7.976,149.460
C08167=1105.678,92.345,-58.281,-179.794,7.980,149.461
C08168=1105.673,92.593,-58.300,-179.793,7.983,149.461
C08169=1105.669,92.843,-58.319,-179.792,7.987,149.462
C08170=1105.663,93.091,-58.338,-179.790,7.991,149.462
C08171=1105.659,93.341,-58.358,-179.789,7.995,149.463
C08172=1105.654,93.590,-58.377,-179.788,7.998,149.463
C08173=1105.649,93.840,-58.395,-179.787,8.003,149.464
C08174=1105.644,94.089,-58.415,-179.785,8.006,149.464
C08175=1105.640,94.338,-58.434,-179.783,8.010,149.465
C08176=1105.635,94.588,-58.454,-179.782,8.013,149.465
C08177=1105.630,94.836,-58.472,-179.781,8.017,149.466
C08178=1105.626,95.086,-58.492,-179.779,8.021,149.466
C08179=1105.620,95.334,-58.511,-179.778,8.025,149.466
C08180=1105.616,95.584,-58.531,-179.777,8.029,149.467
C08181=1105.611,95.833,-58.549,-179.776,8.033,149.467
C08182=1105.606,96.082,-58.569,-179.774,8.036,149.468
C08183=1105.601,96.332,-58.589,-179.772,8.040,149.468
C08184=1105.597,96.580,-58.608,-179.771,8.043,149.469
C08185=1105.592,96.830,-58.627,-179.770,8.047,149.469
C08186=1105.587,97.079,-58.646,-179.768,8.051,149.470
C08187=1105.583,97.328,-58.666,-179.767,8.055,149.470
C08188=1105.578,97.578,-58.685,-179.766,8.058,149.471
C08189=1105.573,97.826,-58.704,-179.764,8.062,149.471
C08190=1105.568,98.076,-58.724,-179.762,8.066,149.471
C08191=1105.564,98.325,-58.743,-179.761,8.070,149.472
C08192=1105.559,98.574,-58.762,-179.759,8.074,149.472
C08193=1105.554,98.824,-58.782,-179.758,8.077,149.473
C08194=1105.548,99.073,-58.801,-179.757,8.081,149.473
C08195=1105.544,99.322,-58.821,-179.755,8.085,149.474
C08196=1105.540,99.571,-58.840,-179.753,8.088,149.474
C08197=1105.534,99.820,-58.859,-179.752,8.092,149.474
C08198=1105.530,100.069,-58.880,-179.751,8.095,149.475
C08199=1105.525,100.319,-58.899,-179.749,8.099,149.475
C08200=1105.520,100.568,-58.919,-179.748,8.103,149.476
C08201=1105.516,100.817,-58.938,-179.746,8.107,149.476
C08202=1105.511,101.066,-58.957,-179.744,8.111,149.477
C08203=1105.506,101.315,-58.977,-179.743,8.114,149.477
C08204=1105.501,101.564,-58.997,-179.741,8.118,149.477
C08205=1105.497,101.814,-59.017,-179.740,8.122,149.478
C08206=1105.492,102.063,-59.036,-179.738,8.125,149.478
C08207=1105.486,102.312,-59.056,-179.737,8.129,149.479
C08208=1105.482,102.562,-59.075,-179.735,8.133,149.479
C08209=1105.478,102.810,-59.095,-179.734,8.136,149.479
C08210=1105.473,103.059,-59.114,-179.732,8.140,149.480
C08211=1105.468,103.309,-59.134,-179.730,8.144,149.480
C08212=1105.464,103.558,-59.154,-179.729,8.148,149.481
C08213=1105.459,103.807,-59.174,-179.727,8.151,149.481
C08214=1105.453,104.056,-59.193,-179.725,8.155,149.481
C08215=1105.449,104.306,-59.213,-179.724,8.158,149.482
C08216=1105.445,104.519,-59.230,-179.722,8.162,149.482
C08217=1105.441,104.733,-59.247,-179.721,8.165,149.482
C08218=1105.437,104.946,-59.264,-179.720,8.167,149.483
C08219=1105.433,105.160,-59.281,-179.718,8.171,149.483
C08220=1105.429,105.373,-59.298,-179.717,8.174,149.483
C08221=1105.424,105.586,-59.315,-179.716,8.177,149.484
C08222=1105.421,105.800,-59.332,-179.714,8.181,149.484
C08223=1105.416,106.013,-59.349,-179.712,8.183,149.484
C08224=1105.412,106.263,-59.369,-179.711,8.187,149.485
C08225=1105.407,106.512,-59.389,-179.709,8.191,149.485
C08226=1105.402,106.761,-59.409,-179.707,8.194,149.485
C08227=1105.397,107.010,-59.429,-179.706,8.198,149.486
C08228=1105.393,107.259,-59.449,-179.704,8.201,149.486
C08229=1105.388,107.508,-59.469,-179.702,8.205,149.486
C08230=1105.384,107.758,-59.489,-179.700,8.209,149.487
C08231=1105.378,108.007,-59.508,-179.699,8.212,149.487
C08232=1105.374,108.256,-59.528,-179.696,8.216,149.487
C08233=1105.369,108.505,-59.548,-179.695,8.220,149.488
C08234=1105.365,108.754,-59.568,-179.693,8.223,149.488
C08235=1105.360,109.003,-59.589,-179.692,8.226,149.488
C08236=1105.355,109.253,-59.609,-179.690,8.230,149.489
C08237=1105.350,109.501,-59.629,-179.688,8.233,149.489
C08238=1105.345,109.751,-59.649,-179.686,8.237,149.489
C08239=1105.340,110.000,-59.669,-179.684,8.241,149.489
C08240=1105.336,110.249,-59.689,-179.682,8.245,149.490
C08241=1105.331,110.498,-59.709,-179.680,8.248,149.490
C08242=1105.327,110.747,-59.729,-179.679,8.251,149.490
C08243=1105.322,110.997,-59.749,-179.677,8.255,149.491
C08244=1105.316,111.245,-59.770,-179.675,8.258,149.491
C08245=1105.312,111.495,-59.789,-179.673,8.262,149.491
C08246=1105.307,111.744,-59.810,-179.672,8.265,149.492
C08247=1105.303,111.993,-59.830,-179.670,8.268,149.492
C08248=1105.298,112.242,-59.850,-179.669,8.272,149.492
C08249=1105.294,112.491,-59.870,-179.667,8.276,149.493
C08250=1105.288,112.741,-59.891,-179.665,8.279,149.493
C08251=1105.284,112.990,-59.911,-179.663,8.282,149.493
C08252=1105.279,113.239,-59.931,-179.661,8.286,149.493
C08253=1105.275,113.488,-59.951,-179.660,8.289,149.494
C08254=1105.269,113.737,-59.972,-179.658,8.293,149.494
C08255=1105.264,113.986,-59.992,-179.656,8.296,149.494
C08256=1105.260,114.235,-60.012,-179.655,8.299,149.495
C08257=1105.255,114.484,-60.032,-179.653,8.303,149.495
C08258=1105.250,114.733,-60.053,-179.651,8.306,149.495
C08259=1105.246,114.982,-60.074,-179.650,8.309,149.496
C08260=1105.241,115.232,-60.093,-179.648,8.313,149.496
C08261=1105.237,115.481,-60.114,-179.646,8.316,149.496
C08262=1105.231,115.730,-60.135,-179.645,8.319,149.497
C08263=1105.227,115.979,-60.155,-179.643,8.323,149.497
C08264=1105.223,116.228,-60.175,-179.641,8.326,149.497
C08265=1105.217,116.477,-60.196,-179.640,8.329,149.497
C08266=1105.213,116.727,-60.216,-179.638,8.333,149.498
C08267=1105.208,116.976,-60.236,-179.636,8.336,149.498
C08268=1105.203,117.225,-60.257,-179.635,8.340,149.498
C08269=1105.199,117.474,-60.278,-179.633,8.343,149.499
C08270=1105.194,117.723,-60.298,-179.631,8.346,149.499
C08271=1105.189,117.972,-60.319,-179.630,8.350,149.499
C08272=1105.185,118.186,-60.336,-179.628,8.353,149.499
C08273=1105.181,118.399,-60.354,-179.626,8.356,149.500
C08274=1105.177,118.613,-60.372,-179.625,8.359,149.500
C08275=1105.173,118.826,-60.390,-179.623,8.361,149.500
C08276=1105.169,119.040,-60.407,-179.622,8.364,149.500
C08277=1105.165,119.253,-60.425,-179.621,8.367,149.501
C08278=1105.162,119.466,-60.442,-179.619,8.369,149.501
C08279=1105.157,119.679,-60.460,-179.617,8.373,149.501
C08280=1105.152,119.929,-60.481,-179.616,8.376,149.501
C08281=1105.148,120.178,-60.501,-179.614,8.380,149.502
C08282=1105.143,120.427,-60.522,-179.612,8.383,149.502
C08283=1105.138,120.676,-60.543,-179.611,8.386,149.502
C08284=1105.134,120.925,-60.563,-179.609,8.390,149.503
C08285=1105.129,121.174,-60.584,-179.607,8.393,149.503
C08286=1105.124,121.423,-60.605,-179.605,8.396,149.503
C08287=1105.119,121.672,-60.625,-179.604,8.400,149.503
C08288=1105.115,121.921,-60.646,-179.602,8.403,149.504
C08289=1105.110,122.170,-60.668,-179.600,8.406,149.504
C08290=1105.105,122.419,-60.688,-179.598,8.409,149.504
C08291=1105.100,122.668,-60.709,-179.597,8.413,149.505
C08292=1105.096,122.918,-60.730,-179.595,8.416,149.505
C08293=1105.091,123.167,-60.751,-179.593,8.419,149.505
C08294=1105.087,123.416,-60.771,-179.591,8.423,149.506
C08295=1105.082,123.665,-60.792,-179.590,8.426,149.506
C08296=1105.078,123.913,-60.813,-179.588,8.430,149.506
C08297=1105.072,124.163,-60.834,-179.586,8.433,149.506
C08298=1105.068,124.412,-60.854,-179.585,8.436,149.507
C08299=1105.063,124.661,-60.875,-179.583,8.440,149.507
C08300=1105.059,124.911,-60.896,-179.581,8.443,149.507
C08301=1105.054,125.159,-60.918,-179.579,8.446,149.507
C08302=1105.050,125.408,-60.938,-179.578,8.450,149.508
C08303=1105.044,125.657,-60.959,-179.576,8.453,149.508
C08304=1105.040,125.906,-60.981,-179.574,8.456,149.508
C08305=1105.035,126.155,-61.001,-179.572,8.459,149.508
C08306=1105.031,126.405,-61.022,-179.570,8.463,149.509
C08307=1105.026,126.654,-61.043,-179.569,8.466,149.509
C08308=1105.021,126.903,-61.065,-179.567,8.470,149.509
C08309=1105.016,127.152,-61.085,-179.565,8.473,149.510
C08310=1105.012,127.401,-61.106,-179.563,8.476,149.510
C08311=1105.007,127.650,-61.128,-179.562,8.480,149.510
C08312=1105.002,127.899,-61.149,-179.560,8.483,149.511
C08313=1104.998,128.148,-61.170,-179.558,8.487,149.511
C08314=1104.993,128.397,-61.191,-179.556,8.489,149.511
C08315=1104.988,128.646,-61.212,-179.555,8.493,149.511
C08316=1104.984,128.895,-61.233,-179.553,8.497,149.512
C08317=1104.979,129.145,-61.254,-179.551,8.499,149.512
C08318=1104.974,129.393,-61.276,-179.549,8.503,149.512
C08319=1104.970,129.642,-61.296,-179.547,8.507,149.513
C08320=1104.964,129.891,-61.317,-179.546,8.510,149.513
C08321=1104.960,130.141,-61.339,-179.544,8.513,149.513
C08322=1104.956,130.390,-61.360,-179.542,8.517,149.513
C08323=1104.951,130.638,-61.381,-179.541,8.520,149.514
C08324=1104.946,130.888,-61.402,-179.539,8.523,149.514
C08325=1104.941,131.137,-61.424,-179.537,8.527,149.514
C08326=1104.937,131.386,-61.445,-179.535,8.530,149.514
C08327=1104.932,131.634,-61.466,-179.534,8.533,149.515
C08328=1104.928,131.848,-61.485,-179.532,8.536,149.515
C08329=1104.924,132.061,-61.503,-179.530,8.539,149.515
C08330=1104.920,132.275,-61.522,-179.529,8.542,149.515
C08331=1104.916,132.488,-61.540,-179.527,8.545,149.516
C08332=1104.912,132.701,-61.558,-179.526,8.548,149.516
C08333=1104.908,132.914,-61.576,-179.524,8.550,149.516
C08334=1104.904,133.128,-61.594,-179.523,8.553,149.516
C08335=1104.900,133.341,-61.613,-179.521,8.556,149.517
C08336=1104.896,133.590,-61.635,-179.519,8.559,149.517
C08337=1104.891,133.839,-61.655,-179.518,8.563,149.517
C08338=1104.886,134.088,-61.677,-179.516,8.567,149.518
C08339=1104.881,134.337,-61.699,-179.514,8.569,149.518
C08340=1104.877,134.587,-61.720,-179.513,8.573,149.518
C08341=1104.872,134.835,-61.742,-179.511,8.577,149.518
C08342=1104.867,135.084,-61.764,-179.509,8.580,149.519
C08343=1104.863,135.334,-61.784,-179.507,8.583,149.519
C08344=1104.858,135.582,-61.806,-179.505,8.587,149.519
C08345=1104.854,135.832,-61.828,-179.503,8.590,149.520
C08346=1104.849,136.080,-61.850,-179.502,8.593,149.520
C08347=1104.844,136.329,-61.871,-179.500,8.597,149.520
C08348=1104.840,136.579,-61.893,-179.498,8.600,149.521
C08349=1104.835,136.827,-61.914,-179.496,8.604,149.521
C08350=1104.830,137.076,-61.936,-179.495,8.606,149.521
C08351=1104.825,137.326,-61.957,-179.493,8.610,149.521
C08352=1104.821,137.574,-61.978,-179.491,8.614,149.522
C08353=1104.817,137.824,-62.001,-179.489,8.617,149.522
C08354=1104.812,138.072,-62.022,-179.488,8.620,149.522
C08355=1104.807,138.321,-62.044,-179.486,8.624,149.523
C08356=1104.803,138.571,-62.065,-179.484,8.627,149.523
C08357=1104.798,138.820,-62.087,-179.482,8.631,149.523
C08358=1104.794,139.069,-62.109,-179.481,8.634,149.523
C08359=1104.789,139.318,-62.131,-179.479,8.637,149.524
C08360=1104.784,139.566,-62.152,-179.477,8.641,149.524
C08361=1104.780,139.816,-62.174,-179.475,8.645,149.524
C08362=1104.775,140.064,-62.196,-179.473,8.648,149.525
C08363=1104.770,140.314,-62.218,-179.472,8.651,149.525
C08364=1104.766,140.562,-62.240,-179.470,8.655,149.525
C08365=1104.761,140.812,-62.262,-179.468,8.658,149.526
C08366=1104.756,141.061,-62.283,-179.467,8.662,149.526
C08367=1104.752,141.310,-62.305,-179.465,8.665,149.526
C08368=1104.747,141.559,-62.327,-179.463,8.668,149.526
C08369=1104.743,141.808,-62.349,-179.461,8.672,149.527
C08370=1104.738,142.057,-62.370,-179.459,8.675,149.527
C08371=1104.733,142.306,-62.393,-179.458,8.679,149.528
C08372=1104.728,142.555,-62.415,-179.456,8.682,149.528
C08373=1104.724,142.804,-62.437,-179.454,8.686,149.528
C08374=1104.719,143.052,-62.459,-179.452,8.690,149.528
C08375=1104.715,143.302,-62.481,-179.451,8.692,149.529
C08376=1104.710,143.550,-62.503,-179.449,8.696,149.529
C08377=1104.706,143.800,-62.525,-179.447,8.700,149.529
C08378=1104.701,144.048,-62.547,-179.445,8.703,149.530
C08379=1104.697,144.298,-62.569,-179.444,8.706,149.530
C08380=1104.692,144.546,-62.590,-179.442,8.710,149.530
C08381=1104.687,144.796,-62.613,-179.440,8.714,149.531
C08382=1104.682,145.045,-62.635,-179.438,8.717,149.531
C08383=1104.678,145.294,-62.657,-179.436,8.721,149.531
C08384=1104.670,145.685,-62.692,-179.433,8.727,149.532
C08385=1104.663,146.075,-62.726,-179.431,8.732,149.532
C08386=1104.655,146.467,-62.761,-179.428,8.737,149.533
C08387=1104.649,146.858,-62.796,-179.425,8.743,149.533
C08388=1104.644,147.107,-62.817,-179.424,8.746,149.534
C08389=1104.639,147.356,-62.841,-179.422,8.749,149.534
C08390=1104.635,147.605,-62.863,-179.420,8.753,149.534
C08391=1104.630,147.854,-62.884,-179.417,8.756,149.534
C08392=1104.626,148.103,-62.907,-179.416,8.760,149.535
C08393=1104.620,148.352,-62.929,-179.414,8.763,149.535
C08394=1104.616,148.601,-62.951,-179.412,8.766,149.535
C08395=1104.612,148.850,-62.974,-179.410,8.770,149.536
C08396=1104.606,149.099,-62.997,-179.409,8.774,149.536
C08397=1104.602,149.348,-63.019,-179.407,8.777,149.536
C08398=1104.597,149.597,-63.040,-179.405,8.780,149.536
C08399=1104.593,149.845,-63.063,-179.403,8.783,149.537
C08400=1104.588,150.095,-63.086,-179.401,8.787,149.537
C08401=1104.584,150.344,-63.107,-179.399,8.790,149.537
C08402=1104.580,150.592,-63.130,-179.397,8.793,149.537
C08403=1104.575,150.842,-63.153,-179.396,8.797,149.538
C08404=1104.570,151.090,-63.175,-179.394,8.801,149.538
C08405=1104.565,151.340,-63.198,-179.392,8.804,149.538
C08406=1104.561,151.588,-63.221,-179.390,8.807,149.539
C08407=1104.556,151.837,-63.242,-179.388,8.810,149.539
C08408=1104.551,152.087,-63.265,-179.386,8.814,149.539
C08409=1104.547,152.335,-63.288,-179.384,8.817,149.539
C08410=1104.542,152.584,-63.309,-179.382,8.820,149.540
C08411=1104.538,152.833,-63.333,-179.380,8.823,149.540
C08412=1104.533,153.082,-63.355,-179.378,8.827,149.540
C08413=1104.528,153.331,-63.378,-179.377,8.830,149.540
C08414=1104.524,153.580,-63.400,-179.375,8.833,149.540
C08415=1104.519,153.829,-63.423,-179.373,8.837,149.541
C08416=1104.288,143.668,-62.566,-179.445,8.700,149.529
C08417=1104.292,143.419,-62.544,-179.447,8.696,149.528
C08418=1104.297,143.170,-62.522,-179.448,8.693,149.528
C08419=1104.301,142.921,-62.500,-179.450,8.689,149.528
C08420=1104.306,142.672,-62.478,-179.452,8.686,149.527
C08421=1104.310,142.423,-62.456,-179.454,8.682,149.527
C08422=1104.315,142.174,-62.435,-179.455,8.679,149.527
C08423=1104.319,141.925,-62.412,-179.457,8.675,149.527
C08424=1104.324,141.676,-62.391,-179.459,8.672,149.526
C08425=1104.328,141.427,-62.369,-179.461,8.668,149.526
C08426=1104.333,141.178,-62.347,-179.463,8.665,149.526
C08427=1104.339,140.930,-62.325,-179.464,8.662,149.525
C08428=1104.343,140.680,-62.303,-179.466,8.658,149.525
C08429=1104.348,140.432,-62.281,-179.468,8.655,149.525
C08430=1104.352,140.182,-62.259,-179.470,8.651,149.524
C08431=1104.357,139.934,-62.237,-179.471,8.648,149.524
C08432=1104.361,139.684,-62.215,-179.473,8.645,149.524
C08433=1104.367,139.435,-62.194,-179.475,8.641,149.524
C08434=1104.371,139.186,-62.172,-179.477,8.637,149.523
C08435=1104.376,138.937,-62.151,-179.478,8.634,149.523
C08436=1104.381,138.688,-62.129,-179.480,8.631,149.523
C08437=1104.385,138.439,-62.107,-179.482,8.627,149.522
C08438=1104.389,138.191,-62.086,-179.484,8.624,149.522
C08439=1104.393,137.941,-62.064,-179.485,8.621,149.522
C08440=1104.398,137.692,-62.043,-179.487,8.617,149.521
C08441=1104.403,137.443,-62.021,-179.489,8.613,149.521
C08442=1104.408,137.194,-61.999,-179.491,8.610,149.521
C08443=1104.412,136.945,-61.977,-179.493,8.607,149.521
C08444=1104.417,136.696,-61.955,-179.494,8.603,149.520
C08445=1104.422,136.447,-61.934,-179.496,8.600,149.520
C08446=1104.427,136.198,-61.913,-179.498,8.596,149.520
C08447=1104.431,135.949,-61.891,-179.499,8.593,149.519
C08448=1104.436,135.700,-61.869,-179.501,8.590,149.519
C08449=1104.440,135.450,-61.848,-179.503,8.586,149.519
C08450=1104.445,135.202,-61.826,-179.505,8.584,149.519
C08451=1104.449,134.953,-61.805,-179.507,8.580,149.518
C08452=1104.454,134.703,-61.783,-179.509,8.576,149.518
C08453=1104.459,134.455,-61.762,-179.511,8.573,149.518
C08454=1104.464,134.206,-61.740,-179.512,8.570,149.517
C08455=1104.468,133.956,-61.719,-179.514,8.566,149.517
C08456=1104.473,133.707,-61.697,-179.516,8.563,149.517
C08457=1104.477,133.459,-61.676,-179.517,8.560,149.516
C08458=1104.482,133.209,-61.655,-179.519,8.556,149.516
C08459=1104.487,132.961,-61.633,-179.521,8.553,149.516
C08460=1104.492,132.712,-61.611,-179.523,8.549,149.516
C08461=1104.497,132.444,-61.589,-179.525,8.546,149.515
C08462=1104.501,132.175,-61.565,-179.527,8.542,149.515
C08463=1104.506,131.907,-61.542,-179.529,8.538,149.515
C08464=1104.512,131.639,-61.520,-179.530,8.534,149.514
C08465=1104.517,131.390,-61.498,-179.532,8.532,149.514
C08466=1104.521,131.142,-61.477,-179.534,8.528,149.514
C08467=1104.525,130.892,-61.456,-179.536,8.525,149.514
C08468=1104.530,130.644,-61.434,-179.537,8.522,149.513
C08469=1104.535,130.394,-61.413,-179.539,8.518,149.513
C08470=1104.539,130.145,-61.392,-179.541,8.515,149.513
C08471=1104.544,129.896,-61.371,-179.543,8.512,149.512
C08472=1104.549,129.647,-61.350,-179.544,8.508,149.512
C08473=1104.554,129.398,-61.328,-179.546,8.505,149.512
C08474=1104.559,129.149,-61.308,-179.548,8.502,149.511
C08475=1104.563,128.900,-61.286,-179.550,8.498,149.511
C08476=1104.568,128.651,-61.265,-179.552,8.495,149.511
C08477=1104.572,128.402,-61.244,-179.554,8.491,149.511
C08478=1104.577,128.153,-61.223,-179.555,8.488,149.510
C08479=1104.582,127.903,-61.201,-179.557,8.485,149.510
C08480=1104.586,127.655,-61.180,-179.559,8.481,149.510
C08481=1104.591,127.405,-61.159,-179.560,8.478,149.509
C08482=1104.596,127.156,-61.138,-179.562,8.475,149.509
C08483=1104.601,126.908,-61.117,-179.564,8.471,149.509
C08484=1104.605,126.658,-61.096,-179.566,8.468,149.509
C08485=1104.610,126.409,-61.075,-179.567,8.465,149.508
C08486=1104.614,126.160,-61.054,-179.569,8.461,149.508
C08487=1104.620,125.911,-61.033,-179.571,8.458,149.508
C08488=1104.624,125.662,-61.012,-179.573,8.455,149.508
C08489=1104.629,125.413,-60.991,-179.574,8.451,149.507
C08490=1104.633,125.164,-60.970,-179.576,8.448,149.507
C08491=1104.638,124.914,-60.949,-179.578,8.445,149.507
C08492=1104.643,124.665,-60.928,-179.580,8.441,149.506
C08493=1104.647,124.417,-60.907,-179.581,8.438,149.506
C08494=1104.652,124.168,-60.886,-179.583,8.435,149.506
C08495=1104.657,123.919,-60.866,-179.585,8.431,149.506
C08496=1104.662,123.669,-60.845,-179.587,8.428,149.505
C08497=1104.666,123.420,-60.823,-179.588,8.425,149.505
C08498=1104.671,123.171,-60.802,-179.590,8.421,149.505
C08499=1104.675,122.922,-60.782,-179.592,8.418,149.504
C08500=1104.680,122.673,-60.761,-179.594,8.415,149.504
C08501=1104.685,122.424,-60.741,-179.595,8.411,149.504
C08502=1104.690,122.175,-60.720,-179.597,8.408,149.504
C08503=1104.694,121.926,-60.699,-179.599,8.405,149.503
C08504=1104.699,121.677,-60.678,-179.601,8.401,149.503
C08505=1104.703,121.427,-60.657,-179.602,8.398,149.503
C08506=1104.708,121.178,-60.636,-179.604,8.395,149.502
C08507=1104.713,120.929,-60.616,-179.606,8.391,149.502
C08508=1104.717,120.680,-60.595,-179.607,8.388,149.502
C08509=1104.722,120.431,-60.574,-179.609,8.385,149.502
C08510=1104.727,120.182,-60.554,-179.611,8.381,149.501
C08511=1104.732,119.933,-60.533,-179.613,8.378,149.501
C08512=1104.736,119.684,-60.512,-179.614,8.374,149.501
C08513=1104.740,119.471,-60.494,-179.616,8.372,149.500
C08514=1104.745,119.257,-60.477,-179.617,8.369,149.500
C08515=1104.748,119.044,-60.459,-179.619,8.366,149.500
C08516=1104.753,118.830,-60.441,-179.621,8.363,149.500
C08517=1104.756,118.617,-60.424,-179.622,8.360,149.499
C08518=1104.760,118.403,-60.406,-179.624,8.357,149.499
C08519=1104.765,118.191,-60.389,-179.625,8.355,149.499
C08520=1104.769,117.977,-60.371,-179.626,8.352,149.499
C08521=1104.773,117.728,-60.351,-179.628,8.348,149.498
C08522=1104.779,117.479,-60.330,-179.630,8.345,149.498
C08523=1104.783,117.230,-60.310,-179.631,8.342,149.498
C08524=1104.787,116.981,-60.289,-179.633,8.338,149.497
C08525=1104.793,116.732,-60.268,-179.635,8.334,149.497
C08526=1104.797,116.483,-60.248,-179.637,8.332,149.497
C08527=1104.802,116.233,-60.228,-179.638,8.328,149.497
C08528=1104.807,115.984,-60.207,-179.640,8.324,149.496
C08529=1104.811,115.735,-60.187,-179.642,8.322,149.496
C08530=1104.816,115.486,-60.167,-179.643,8.318,149.496
C08531=1104.820,115.237,-60.146,-179.645,8.314,149.495
C08532=1104.825,114.988,-60.125,-179.647,8.312,149.495
C08533=1104.830,114.739,-60.105,-179.648,8.308,149.495
C08534=1104.835,114.489,-60.085,-179.650,8.304,149.495
C08535=1104.840,114.240,-60.064,-179.651,8.301,149.494
C08536=1104.844,113.991,-60.044,-179.654,8.298,149.494
C08537=1104.849,113.742,-60.023,-179.656,8.294,149.494
C08538=1104.853,113.493,-60.004,-179.657,8.291,149.493
C08539=1104.859,113.243,-59.983,-179.659,8.287,149.493
C08540=1104.863,112.994,-59.962,-179.661,8.284,149.493
C08541=1104.867,112.746,-59.942,-179.662,8.281,149.492
C08542=1104.872,112.496,-59.922,-179.664,8.277,149.492
C08543=1104.877,112.247,-59.902,-179.665,8.274,149.492
C08544=1104.882,111.998,-59.881,-179.667,8.271,149.491
C08545=1104.887,111.749,-59.862,-179.669,8.267,149.491
C08546=1104.892,111.500,-59.841,-179.670,8.263,149.491
C08547=1104.896,111.251,-59.821,-179.672,8.261,149.491
C08548=1104.901,111.001,-59.801,-179.674,8.257,149.490
C08549=1104.905,110.752,-59.781,-179.676,8.253,149.490
C08550=1104.910,110.503,-59.760,-179.678,8.250,149.490
C08551=1104.915,110.254,-59.740,-179.679,8.246,149.489
C08552=1104.920,110.005,-59.720,-179.681,8.242,149.489
C08553=1104.925,109.756,-59.701,-179.683,8.239,149.489
C08554=1104.929,109.507,-59.680,-179.684,8.236,149.488
C08555=1104.934,109.258,-59.660,-179.686,8.232,149.488
C08556=1104.939,109.008,-59.640,-179.688,8.228,149.488
C08557=1104.943,108.759,-59.620,-179.690,8.225,149.487
C08558=1104.948,108.510,-59.600,-179.692,8.221,149.487
C08559=1104.954,108.261,-59.580,-179.694,8.218,149.487
C08560=1104.958,108.012,-59.560,-179.695,8.214,149.486
C08561=1104.963,107.763,-59.540,-179.697,8.211,149.486
C08562=1104.967,107.513,-59.520,-179.698,8.207,149.486
C08563=1104.972,107.264,-59.500,-179.700,8.204,149.485
C08564=1104.977,107.015,-59.480,-179.702,8.200,149.485
C08565=1104.982,106.766,-59.460,-179.704,8.196,149.485
C08566=1104.986,106.517,-59.440,-179.706,8.192,149.484
C08567=1104.991,106.267,-59.421,-179.708,8.189,149.484
C08568=1104.996,106.018,-59.400,-179.709,8.186,149.484
C08569=1105.000,105.806,-59.384,-179.711,8.182,149.483
C08570=1105.004,105.592,-59.366,-179.712,8.179,149.483
C08571=1105.007,105.378,-59.350,-179.713,8.176,149.483
C08572=1105.012,105.165,-59.332,-179.715,8.172,149.482
C08573=1105.016,104.952,-59.316,-179.716,8.170,149.482
C08574=1105.020,104.738,-59.298,-179.717,8.167,149.482
C08575=1105.024,104.525,-59.282,-179.719,8.164,149.481
C08576=1105.028,104.310,-59.265,-179.720,8.160,149.481
C08577=1105.033,104.062,-59.245,-179.722,8.157,149.481
C08578=1105.038,103.812,-59.225,-179.723,8.153,149.480
C08579=1105.043,103.563,-59.206,-179.725,8.150,149.480
C08580=1105.048,103.314,-59.186,-179.727,8.146,149.480
C08581=1105.052,103.065,-59.166,-179.729,8.142,149.479
C08582=1105.057,102.815,-59.146,-179.730,8.138,149.479
C08583=1105.061,102.567,-59.126,-179.732,8.134,149.478
C08584=1105.066,102.318,-59.107,-179.733,8.131,149.478
C08585=1105.071,102.068,-59.087,-179.734,8.127,149.478
C08586=1105.076,101.819,-59.068,-179.736,8.124,149.477
C08587=1105.080,101.570,-59.047,-179.738,8.120,149.477
C08588=1105.085,101.321,-59.028,-179.740,8.116,149.476
C08589=1105.090,101.071,-59.008,-179.741,8.113,149.476
C08590=1105.095,100.822,-58.989,-179.742,8.109,149.476
C08591=1105.100,100.573,-58.970,-179.744,8.105,149.475
C08592=1105.104,100.324,-58.950,-179.745,8.101,149.475
C08593=1105.109,100.075,-58.930,-179.747,8.097,149.474
C08594=1105.114,99.826,-58.911,-179.748,8.095,149.474
C08595=1105.119,99.576,-58.891,-179.750,8.091,149.474
C08596=1105.123,99.327,-58.872,-179.752,8.087,149.473
C08597=1105.128,99.078,-58.853,-179.753,8.083,149.473
C08598=1105.133,98.829,-58.833,-179.755,8.079,149.472
C08599=1105.138,98.579,-58.814,-179.756,8.076,149.472
C08600=1105.143,98.330,-58.794,-179.757,8.072,149.471
C08601=1105.147,98.081,-58.774,-179.759,8.068,149.471
C08602=1105.152,97.833,-58.755,-179.761,8.064,149.471
C08603=1105.157,97.583,-58.735,-179.762,8.061,149.470
C08604=1105.162,97.333,-58.716,-179.763,8.057,149.470
C08605=1105.166,97.085,-58.697,-179.764,8.053,149.469
C08606=1105.171,96.835,-58.677,-179.766,8.049,149.469
C08607=1105.176,96.586,-58.658,-179.768,8.045,149.468
C08608=1105.181,96.337,-58.639,-179.769,8.042,149.468
C08609=1105.185,96.088,-58.619,-179.770,8.038,149.467
C08610=1105.190,95.839,-58.600,-179.772,8.035,149.467
C08611=1105.195,95.589,-58.581,-179.773,8.031,149.466
C08612=1105.199,95.340,-58.561,-179.774,8.028,149.466
C08613=1105.204,95.091,-58.542,-179.776,8.024,149.466
C08614=1105.209,94.841,-58.523,-179.777,8.019,149.465
C08615=1105.214,94.592,-58.505,-179.779,8.015,149.464
C08616=1105.219,94.343,-58.485,-179.780,8.012,149.464
C08617=1105.224,94.094,-58.466,-179.781,8.008,149.464
C08618=1105.228,93.845,-58.447,-179.783,8.005,149.463
C08619=1105.233,93.595,-58.427,-179.784,8.001,149.463
C08620=1105.238,93.346,-58.408,-179.785,7.997,149.462
C08621=1105.242,93.097,-58.389,-179.787,7.993,149.462
C08622=1105.248,92.848,-58.369,-179.788,7.989,149.461
C08623=1105.253,92.598,-58.350,-179.789,7.986,149.461
C08624=1105.257,92.349,-58.332,-179.790,7.982,149.460
C08625=1105.261,92.136,-58.315,-179.792,7.979,149.460
C08626=1105.266,91.922,-58.298,-179.793,7.975,149.459
C08627=1105.269,91.709,-58.282,-179.794,7.972,149.459
C08628=1105.274,91.495,-58.266,-179.795,7.969,149.459
C08629=1105.278,91.281,-58.250,-179.796,7.966,149.458
C08630=1105.282,91.068,-58.233,-179.797,7.963,149.458
C08631=1105.286,90.854,-58.217,-179.798,7.960,149.457
C08632=1105.290,90.641,-58.200,-179.800,7.956,149.457
C08633=1105.295,90.391,-58.182,-179.801,7.953,149.456
C08634=1105.300,90.143,-58.163,-179.802,7.949,149.456
C08635=1105.304,89.893,-58.144,-179.803,7.945,149.455
C08636=1105.309,89.644,-58.124,-179.804,7.942,149.455
C08637=1105.314,89.395,-58.106,-179.805,7.937,149.454
C08638=1105.319,89.146,-58.087,-179.807,7.933,149.454
C08639=1105.323,88.896,-58.068,-179.808,7.930,149.453
C08640=1105.329,88.647,-58.049,-179.809,7.926,149.453
C08641=1105.333,88.398,-58.030,-179.811,7.922,149.452
C08642=1105.338,88.149,-58.011,-179.812,7.919,149.452
C08643=1105.342,87.899,-57.992,-179.813,7.915,149.451
C08644=1105.348,87.650,-57.973,-179.814,7.911,149.451
C08645=1105.352,87.401,-57.954,-179.815,7.907,149.450
C08646=1105.357,87.151,-57.935,-179.817,7.904,149.450
C08647=1105.362,86.903,-57.917,-179.818,7.900,149.449
C08648=1105.367,86.653,-57.898,-179.819,7.896,149.449
C08649=1105.372,86.404,-57.879,-179.820,7.892,149.448
C08650=1105.376,86.155,-57.860,-179.821,7.889,149.447
C08651=1105.381,85.905,-57.841,-179.822,7.885,149.447
C08652=1105.385,85.656,-57.822,-179.824,7.881,149.446
C08653=1105.391,85.407,-57.804,-179.824,7.877,149.446
C08654=1105.396,85.158,-57.785,-179.826,7.874,149.446
C08655=1105.400,84.908,-57.767,-179.827,7.870,149.445
C08656=1105.405,84.659,-57.747,-179.828,7.866,149.444
C08657=1105.410,84.409,-57.729,-179.829,7.862,149.444
C08658=1105.415,84.160,-57.710,-179.830,7.859,149.443
C08659=1105.420,83.911,-57.692,-179.831,7.855,149.443
C08660=1105.424,83.662,-57.673,-179.832,7.851,149.442
C08661=1105.430,83.413,-57.654,-179.833,7.847,149.442
C08662=1105.434,83.164,-57.635,-179.834,7.844,149.441
C08663=1105.438,82.914,-57.617,-179.836,7.840,149.441
C08664=1105.444,82.665,-57.598,-179.837,7.836,149.440
C08665=1105.449,82.416,-57.580,-179.838,7.832,149.439
C08666=1105.453,82.166,-57.561,-179.839,7.828,149.439
C08667=1105.458,81.917,-57.542,-179.840,7.825,149.438
C08668=1105.463,81.667,-57.524,-179.841,7.821,149.438
C08669=1105.467,81.419,-57.505,-179.842,7.818,149.437
C08670=1105.473,81.169,-57.487,-179.843,7.814,149.437
C08671=1105.477,80.920,-57.468,-179.844,7.810,149.436
C08672=1105.482,80.671,-57.450,-179.846,7.806,149.436
C08673=1105.487,80.422,-57.432,-179.846,7.803,149.435
C08674=1105.492,80.172,-57.413,-179.848,7.799,149.435
C08675=1105.496,79.923,-57.394,-179.848,7.795,149.434
C08676=1105.501,79.674,-57.376,-179.849,7.791,149.433
C08677=1105.507,79.424,-57.357,-179.850,7.788,149.433
C08678=1105.511,79.175,-57.338,-179.851,7.784,149.432
C08679=1105.516,78.926,-57.320,-179.852,7.781,149.432
C08680=1105.521,78.677,-57.302,-179.853,7.776,149.431
C08681=1105.525,78.463,-57.286,-179.854,7.773,149.431
C08682=1105.529,78.249,-57.271,-179.855,7.770,149.430
C08683=1105.533,78.036,-57.255,-179.856,7.767,149.430
C08684=1105.537,77.822,-57.239,-179.857,7.764,149.429
C08685=1105.542,77.608,-57.223,-179.858,7.760,149.429
C08686=1105.546,77.395,-57.207,-179.859,7.757,149.428
C08687=1105.550,77.181,-57.191,-179.860,7.754,149.428
C08688=1105.554,76.968,-57.176,-179.861,7.751,149.428
C08689=1105.559,76.718,-57.157,-179.862,7.747,149.427
C08690=1105.564,76.468,-57.139,-179.863,7.744,149.426
C08691=1105.568,76.219,-57.121,-179.864,7.740,149.426
C08692=1105.573,75.971,-57.102,-179.865,7.735,149.425
C08693=1105.578,75.722,-57.084,-179.867,7.732,149.425
C08694=1105.582,75.472,-57.066,-179.869,7.728,149.424
C08695=1105.588,75.222,-57.047,-179.870,7.724,149.424
C08696=1105.593,74.973,-57.030,-179.871,7.720,149.423
C08697=1105.598,74.724,-57.012,-179.873,7.716,149.423
C08698=1105.602,74.475,-56.992,-179.874,7.712,149.423
C08699=1105.607,74.225,-56.974,-179.876,7.707,149.422
C08700=1105.612,73.976,-56.957,-179.877,7.704,149.421
C08701=1105.617,73.727,-56.939,-179.878,7.700,149.421
C08702=1105.621,73.478,-56.921,-179.879,7.696,149.420
C08703=1105.626,73.228,-56.902,-179.881,7.692,149.420
C08704=1105.631,72.979,-56.884,-179.882,7.688,149.419
C08705=1105.636,72.729,-56.866,-179.884,7.684,149.419
C08706=1105.641,72.480,-56.848,-179.885,7.680,149.418
C08707=1105.646,72.231,-56.830,-179.887,7.676,149.418
C08708=1105.651,71.982,-56.812,-179.888,7.672,149.418
C08709=1105.655,71.732,-56.793,-179.889,7.669,149.417
C08710=1105.660,71.483,-56.775,-179.890,7.665,149.416
C08711=1105.665,71.234,-56.757,-179.892,7.661,149.416
C08712=1105.670,70.984,-56.739,-179.893,7.657,149.415
C08713=1105.675,70.735,-56.721,-179.895,7.653,149.415
C08714=1105.680,70.486,-56.703,-179.896,7.649,149.414
C08715=1105.685,70.237,-56.685,-179.897,7.645,149.414
C08716=1105.689,69.987,-56.667,-179.899,7.641,149.413
C08717=1105.694,69.738,-56.649,-179.900,7.638,149.413
C08718=1105.699,69.489,-56.631,-179.901,7.633,149.412
C08719=1105.704,69.240,-56.613,-179.902,7.629,149.412
C08720=1105.709,68.990,-56.596,-179.904,7.625,149.411
C08721=1105.714,68.741,-56.578,-179.905,7.621,149.411
C08722=1105.719,68.491,-56.560,-179.907,7.617,149.410
C08723=1105.724,68.242,-56.542,-179.908,7.613,149.410
C08724=1105.728,67.993,-56.525,-179.909,7.610,149.409
C08725=1105.732,67.743,-56.506,-179.910,7.606,149.409
C08726=1105.737,67.494,-56.488,-179.911,7.602,149.408
C08727=1105.742,67.244,-56.471,-179.913,7.598,149.408
C08728=1105.747,66.995,-56.453,-179.914,7.594,149.407
C08729=1105.752,66.746,-56.435,-179.916,7.590,149.407
C08730=1105.757,66.497,-56.417,-179.917,7.587,149.406
C08731=1105.762,66.247,-56.400,-179.918,7.582,149.406
C08732=1105.767,65.998,-56.382,-179.919,7.578,149.405
C08733=1105.771,65.749,-56.364,-179.920,7.574,149.404
C08734=1105.776,65.500,-56.346,-179.922,7.570,149.404
C08735=1105.782,65.250,-56.329,-179.923,7.566,149.404
C08736=1105.787,65.001,-56.311,-179.924,7.563,149.403
C08737=1105.791,64.788,-56.295,-179.926,7.559,149.403
C08738=1105.794,64.573,-56.281,-179.926,7.556,149.402
C08739=1105.799,64.359,-56.266,-179.927,7.553,149.402
C08740=1105.803,64.146,-56.251,-179.929,7.549,149.401
C08741=1105.807,63.932,-56.236,-179.930,7.546,149.401
C08742=1105.811,63.719,-56.220,-179.931,7.542,149.400
C08743=1105.816,63.505,-56.205,-179.932,7.539,149.400
C08744=1105.819,63.291,-56.191,-179.933,7.535,149.399
C08745=1105.824,63.041,-56.173,-179.934,7.531,149.399
C08746=1105.829,62.792,-56.155,-179.935,7.528,149.398
C08747=1105.834,62.542,-56.137,-179.937,7.524,149.398
C08748=1105.838,62.294,-56.120,-179.938,7.520,149.397
C08749=1105.843,62.044,-56.102,-179.939,7.516,149.397
C08750=1105.849,61.795,-56.085,-179.941,7.512,149.396
C08751=1105.853,61.545,-56.067,-179.941,7.508,149.396
C08752=1105.858,61.296,-56.050,-179.943,7.504,149.395
C08753=1105.863,61.047,-56.032,-179.944,7.500,149.394
C08754=1105.869,60.798,-56.015,-179.945,7.496,149.394
C08755=1105.874,60.548,-55.997,-179.947,7.492,149.393
C08756=1105.878,60.299,-55.981,-179.948,7.489,149.393
C08757=1105.883,60.050,-55.963,-179.949,7.484,149.392
C08758=1105.888,59.800,-55.945,-179.950,7.480,149.392
C08759=1105.892,59.551,-55.928,-179.951,7.476,149.391
C08760=1105.898,59.301,-55.911,-179.953,7.472,149.391
C08761=1105.903,59.052,-55.893,-179.953,7.469,149.390
C08762=1105.907,58.803,-55.876,-179.955,7.465,149.390
C08763=1105.912,58.554,-55.858,-179.956,7.461,149.389
C08764=1105.917,58.304,-55.841,-179.958,7.457,149.389
C08765=1105.921,58.055,-55.823,-179.959,7.452,149.388
C08766=1105.927,57.806,-55.806,-179.960,7.449,149.387
C08767=1105.932,57.556,-55.789,-179.961,7.445,149.387
C08768=1105.937,57.307,-55.772,-179.962,7.441,149.386
C08769=1105.942,57.057,-55.755,-179.963,7.437,149.386
C08770=1105.946,56.808,-55.737,-179.965,7.433,149.385
C08771=1105.951,56.559,-55.720,-179.965,7.429,149.385
C08772=1105.956,56.309,-55.703,-179.966,7.425,149.384
C08773=1105.961,56.060,-55.685,-179.968,7.421,149.384
C08774=1105.966,55.811,-55.668,-179.969,7.417,149.383
C08775=1105.971,55.561,-55.652,-179.970,7.414,149.382
C08776=1105.976,55.312,-55.634,-179.971,7.409,149.382
C08777=1105.981,55.062,-55.616,-179.973,7.405,149.381
C08778=1105.985,54.813,-55.600,-179.974,7.401,149.381
C08779=1105.990,54.564,-55.582,-179.975,7.397,149.380
C08780=1105.995,54.314,-55.565,-179.976,7.394,149.380
C08781=1106.001,54.065,-55.548,-179.977,7.389,149.379
C08782=1106.005,53.816,-55.532,-179.978,7.386,149.379
C08783=1106.010,53.567,-55.514,-179.980,7.381,149.378
C08784=1106.015,53.317,-55.497,-179.980,7.378,149.377
C08785=1106.020,53.067,-55.480,-179.982,7.374,149.377
C08786=1106.025,52.819,-55.463,-179.983,7.370,149.376
C08787=1106.030,52.569,-55.446,-179.984,7.365,149.376
C08788=1106.034,52.320,-55.429,-179.985,7.362,149.375
C08789=1106.039,52.070,-55.411,-179.986,7.358,149.374
C08790=1106.044,51.821,-55.395,-179.987,7.354,149.374
C08791=1106.050,51.571,-55.378,-179.988,7.350,149.373
C08792=1106.054,51.322,-55.361,-179.989,7.346,149.373
C08793=1106.059,51.108,-55.346,-179.990,7.342,149.372
C08794=1106.063,50.894,-55.332,-179.991,7.339,149.372
C08795=1106.067,50.681,-55.317,-179.992,7.336,149.371
C08796=1106.071,50.467,-55.303,-179.993,7.332,149.371
C08797=1106.076,50.253,-55.288,-179.994,7.329,149.370
C08798=1106.080,50.039,-55.273,-179.995,7.325,149.370
C08799=1106.084,49.825,-55.259,-179.996,7.322,149.369
C08800=1106.088,49.612,-55.245,-179.997,7.319,149.369
C08801=1106.093,49.362,-55.227,-179.998,7.314,149.368
C08802=1106.097,49.112,-55.211,-179.999,7.310,149.367
C08803=1106.102,48.864,-55.194,-180.000,7.307,149.367
C08804=1106.108,48.614,-55.177,179.999,7.303,149.366
C08805=1106.112,48.364,-55.160,179.998,7.298,149.366
C08806=1106.118,48.115,-55.144,179.997,7.294,149.365
C08807=1106.122,47.866,-55.127,179.996,7.291,149.365
C08808=1106.127,47.616,-55.110,179.995,7.287,149.364
C08809=1106.132,47.367,-55.093,179.994,7.282,149.363
C08810=1106.137,47.118,-55.077,179.993,7.278,149.363
C08811=1106.142,46.868,-55.060,179.992,7.275,149.362
C08812=1106.147,46.618,-55.043,179.991,7.271,149.362
C08813=1106.152,46.370,-55.026,179.990,7.266,149.361
C08814=1106.156,46.120,-55.010,179.989,7.262,149.360
C08815=1106.161,45.871,-54.993,179.988,7.259,149.360
C08816=1106.167,45.622,-54.976,179.987,7.255,149.359
C08817=1106.171,45.372,-54.960,179.986,7.250,149.359
C08818=1106.176,45.122,-54.944,179.984,7.246,149.358
C08819=1106.182,44.873,-54.927,179.984,7.243,149.357
C08820=1106.186,44.623,-54.910,179.982,7.239,149.357
C08821=1106.191,44.374,-54.893,179.981,7.234,149.356
C08822=1106.196,44.125,-54.877,179.980,7.230,149.355
C08823=1106.201,43.875,-54.860,179.980,7.227,149.355
C08824=1106.206,43.626,-54.843,179.979,7.222,149.354
C08825=1106.211,43.377,-54.827,179.978,7.218,149.353
C08826=1106.215,43.127,-54.811,179.976,7.214,149.353
C08827=1106.221,42.877,-54.794,179.976,7.211,149.352
C08828=1106.226,42.628,-54.777,179.975,7.206,149.352
C08829=1106.230,42.379,-54.761,179.974,7.202,149.351
C08830=1106.235,42.130,-54.744,179.973,7.198,149.350
C08831=1106.240,41.880,-54.728,179.972,7.194,149.350
C08832=1106.245,41.630,-54.711,179.971,7.190,149.349
C08833=1106.250,41.382,-54.695,179.970,7.185,149.348
C08834=1106.255,41.132,-54.678,179.969,7.182,149.348
C08835=1106.260,40.883,-54.663,179.968,7.178,149.347
C08836=1106.265,40.633,-54.646,179.967,7.174,149.347
C08837=1106.269,40.384,-54.629,179.966,7.169,149.346
C08838=1106.275,40.134,-54.613,179.965,7.166,149.345
C08839=1106.280,39.884,-54.596,179.964,7.162,149.345
C08840=1106.285,39.636,-54.580,179.963,7.157,149.344
C08841=1106.289,39.386,-54.563,179.963,7.154,149.343
C08842=1106.295,39.137,-54.548,179.962,7.150,149.343
C08843=1106.299,38.887,-54.531,179.961,7.145,149.342
C08844=1106.304,38.638,-54.514,179.959,7.141,149.341
C08845=1106.310,38.388,-54.498,179.959,7.137,149.341
C08846=1106.314,38.139,-54.482,179.958,7.133,149.340
C08847=1106.320,37.889,-54.466,179.957,7.129,149.340
C08848=1106.324,37.640,-54.449,179.956,7.125,149.339
C08849=1106.328,37.425,-54.436,179.955,7.121,149.338
C08850=1106.333,37.212,-54.422,179.954,7.118,149.338
C08851=1106.337,36.998,-54.408,179.954,7.114,149.337
C08852=1106.341,36.784,-54.393,179.953,7.111,149.337
C08853=1106.346,36.570,-54.380,179.953,7.108,149.336
C08854=1106.350,36.356,-54.365,179.951,7.104,149.336
C08855=1106.354,36.143,-54.352,179.951,7.100,149.335
C08856=1106.358,35.929,-54.339,179.950,7.097,149.334
C08857=1106.363,35.679,-54.322,179.949,7.092,149.334
C08858=1106.369,35.430,-54.306,179.949,7.089,149.333
C08859=1106.373,35.180,-54.289,179.948,7.085,149.332
C08860=1106.379,34.931,-54.274,179.947,7.080,149.332
C08861=1106.383,34.681,-54.257,179.945,7.076,149.331
C08862=1106.388,34.432,-54.241,179.945,7.072,149.330
C08863=1106.393,34.182,-54.225,179.944,7.068,149.330
C08864=1106.398,33.933,-54.209,179.943,7.064,149.329
C08865=1106.403,33.684,-54.193,179.942,7.060,149.328
C08866=1106.408,33.434,-54.177,179.941,7.056,149.328
C08867=1106.413,33.185,-54.161,179.941,7.051,149.327
C08868=1106.418,32.935,-54.145,179.940,7.047,149.326
C08869=1106.422,32.687,-54.129,179.939,7.043,149.326
C08870=1106.427,32.437,-54.113,179.938,7.039,149.325
C08871=1106.432,32.187,-54.097,179.937,7.035,149.324
C08872=1106.437,31.938,-54.081,179.937,7.031,149.324
C08873=1106.442,31.688,-54.065,179.936,7.027,149.323
C08874=1106.447,31.439,-54.049,179.935,7.022,149.322
C08875=1106.452,31.189,-54.033,179.934,7.018,149.321
C08876=1106.458,30.940,-54.017,179.934,7.015,149.321
C08877=1106.462,30.690,-54.001,179.933,7.010,149.320
C08878=1106.467,30.441,-53.985,179.931,7.006,149.319
C08879=1106.472,30.191,-53.969,179.931,7.002,149.318
C08880=1106.477,29.943,-53.953,179.930,6.998,149.318
C08881=1106.482,29.693,-53.938,179.929,6.993,149.317
C08882=1106.487,29.443,-53.922,179.928,6.989,149.317
C08883=1106.492,29.194,-53.906,179.928,6.985,149.316
C08884=1106.497,28.945,-53.890,179.927,6.981,149.315
C08885=1106.502,28.695,-53.874,179.926,6.977,149.314
C08886=1106.507,28.445,-53.858,179.926,6.973,149.314
C08887=1106.511,28.196,-53.842,179.925,6.968,149.313
C08888=1106.517,27.947,-53.827,179.924,6.964,149.312
C08889=1106.522,27.697,-53.811,179.923,6.960,149.311
C08890=1106.527,27.447,-53.795,179.923,6.956,149.311
C08891=1106.532,27.198,-53.779,179.922,6.952,149.310
C08892=1106.537,26.949,-53.763,179.921,6.947,149.309
C08893=1106.541,26.699,-53.748,179.921,6.943,149.308
C08894=1106.547,26.450,-53.732,179.920,6.939,149.308
C08895=1106.552,26.200,-53.717,179.919,6.935,149.307
C08896=1106.556,25.951,-53.700,179.918,6.930,149.306
C08897=1106.561,25.702,-53.685,179.918,6.926,149.306
C08898=1106.567,25.452,-53.670,179.917,6.922,149.305
C08899=1106.571,25.202,-53.654,179.916,6.917,149.304
C08900=1106.577,24.953,-53.638,179.916,6.914,149.303
C08901=1106.582,24.704,-53.622,179.915,6.910,149.303
C08902=1106.586,24.454,-53.607,179.914,6.905,149.302
C08903=1106.591,24.205,-53.591,179.913,6.901,149.301
C08904=1106.597,23.956,-53.575,179.913,6.897,149.300
C08905=1106.600,23.742,-53.562,179.913,6.893,149.300
C08906=1106.605,23.528,-53.549,179.911,6.889,149.299
C08907=1106.609,23.314,-53.535,179.911,6.886,149.299
C08908=1106.613,23.099,-53.523,179.910,6.882,149.298
C08909=1106.618,22.885,-53.509,179.910,6.879,149.297
C08910=1106.622,22.671,-53.496,179.910,6.875,149.297
C08911=1106.626,22.457,-53.482,179.909,6.871,149.296
C08912=1106.631,22.243,-53.469,179.908,6.867,149.295
C08913=1106.636,21.993,-53.453,179.908,6.863,149.294
C08914=1106.640,21.744,-53.438,179.907,6.859,149.294
C08915=1106.646,21.495,-53.423,179.907,6.854,149.293
C08916=1106.651,21.245,-53.407,179.905,6.850,149.292
C08917=1106.655,20.996,-53.392,179.906,6.846,149.291
C08918=1106.660,20.746,-53.376,179.904,6.842,149.291
C08919=1106.666,20.497,-53.360,179.904,6.837,149.290
C08920=1106.671,20.248,-53.345,179.903,6.834,149.289
C08921=1106.675,19.998,-53.330,179.903,6.829,149.288
C08922=1106.680,19.749,-53.315,179.902,6.825,149.287
C08923=1106.685,19.499,-53.299,179.901,6.820,149.287
C08924=1106.691,19.250,-53.283,179.901,6.816,149.286
C08925=1106.695,19.000,-53.268,179.900,6.812,149.285
C08926=1106.700,18.751,-53.252,179.900,6.807,149.284
C08927=1106.705,18.501,-53.237,179.899,6.803,149.284
C08928=1106.710,18.252,-53.222,179.899,6.799,149.283
C08929=1106.716,18.002,-53.207,179.898,6.794,149.282
C08930=1106.720,17.752,-53.192,179.897,6.790,149.281
C08931=1106.725,17.503,-53.176,179.897,6.786,149.280
C08932=1106.730,17.254,-53.161,179.897,6.781,149.279
C08933=1106.735,17.004,-53.145,179.896,6.777,149.279
C08934=1106.740,16.755,-53.130,179.895,6.772,149.278
C08935=1106.745,16.506,-53.115,179.895,6.768,149.277
C08936=1106.750,16.255,-53.100,179.894,6.764,149.276
C08937=1106.755,16.006,-53.085,179.893,6.759,149.275
C08938=1106.761,15.757,-53.069,179.893,6.754,149.274
C08939=1106.765,15.508,-53.054,179.892,6.751,149.274
C08940=1106.771,15.258,-53.038,179.892,6.746,149.273
C08941=1106.776,15.008,-53.024,179.891,6.742,149.272
C08942=1106.780,14.759,-53.009,179.891,6.738,149.271
C08943=1106.785,14.509,-52.993,179.890,6.733,149.270
C08944=1106.790,14.260,-52.978,179.890,6.729,149.270
C08945=1106.795,14.010,-52.963,179.889,6.724,149.269
C08946=1106.800,13.761,-52.948,179.889,6.720,149.268
C08947=1106.805,13.512,-52.933,179.888,6.716,149.267
C08948=1106.810,13.262,-52.919,179.888,6.711,149.266
C08949=1106.816,13.013,-52.903,179.887,6.706,149.265
C08950=1106.820,12.763,-52.888,179.887,6.702,149.265
C08951=1106.825,12.513,-52.872,179.887,6.698,149.264
C08952=1106.830,12.264,-52.858,179.886,6.693,149.263
C08953=1106.835,12.015,-52.843,179.885,6.689,149.262
C08954=1106.840,11.765,-52.827,179.885,6.685,149.261
C08955=1106.845,11.515,-52.813,179.885,6.680,149.260
C08956=1106.850,11.266,-52.797,179.884,6.675,149.259
C08957=1106.855,11.016,-52.783,179.884,6.671,149.259
C08958=1106.861,10.767,-52.767,179.884,6.667,149.258
C08959=1106.865,10.518,-52.752,179.883,6.662,149.257
C08960=1106.870,10.268,-52.738,179.882,6.657,149.256
C08961=1106.875,10.054,-52.724,179.882,6.654,149.255
C08962=1106.879,9.840,-52.712,179.882,6.650,149.255
C08963=1106.883,9.626,-52.699,179.882,6.646,149.254
C08964=1106.888,9.412,-52.687,179.881,6.642,149.253
C08965=1106.891,9.198,-52.674,179.880,6.638,149.252
C08966=1106.897,8.983,-52.661,179.880,6.635,149.251
C08967=1106.900,8.769,-52.648,179.880,6.631,149.251
C08968=1106.905,8.555,-52.636,179.880,6.627,149.250
C08969=1106.910,8.306,-52.620,179.879,6.623,149.249
C08970=1106.915,8.056,-52.606,179.878,6.618,149.248
C08971=1106.920,7.807,-52.591,179.878,6.613,149.247
C08972=1106.925,7.557,-52.576,179.877,6.608,149.247
C08973=1106.930,7.308,-52.561,179.876,6.603,149.246
C08974=1106.935,7.058,-52.547,179.875,6.599,149.245
C08975=1106.940,6.809,-52.531,179.875,6.594,149.244
C08976=1106.945,6.559,-52.517,179.874,6.589,149.243
C08977=1106.950,6.310,-52.502,179.874,6.585,149.242
C08978=1106.955,6.060,-52.488,179.873,6.581,149.242
C08979=1106.960,5.811,-52.472,179.873,6.576,149.241
C08980=1106.965,5.561,-52.458,179.872,6.572,149.240
C08981=1106.970,5.312,-52.443,179.872,6.567,149.239
C08982=1106.975,5.063,-52.428,179.871,6.562,149.238
C08983=1106.981,4.813,-52.414,179.870,6.558,149.237
C08984=1106.985,4.563,-52.399,179.869,6.553,149.237
C08985=1106.990,4.314,-52.384,179.869,6.549,149.236
C08986=1106.995,4.064,-52.370,179.868,6.544,149.235
C08987=1107.000,3.815,-52.355,179.867,6.540,149.234
C08988=1107.005,3.565,-52.340,179.867,6.535,149.233
C08989=1107.010,3.315,-52.326,179.866,6.530,149.232
C08990=1107.015,3.066,-52.311,179.865,6.526,149.232
C08991=1107.020,2.816,-52.297,179.865,6.521,149.231
C08992=1107.025,2.567,-52.282,179.864,6.516,149.230
C08993=1107.030,2.317,-52.267,179.864,6.512,149.229
C08994=1107.035,2.068,-52.253,179.863,6.507,149.228
C08995=1107.040,1.818,-52.238,179.862,6.503,149.227
C08996=1107.045,1.568,-52.224,179.862,6.498,149.227
C08997=1107.050,1.320,-52.209,179.861,6.493,149.226
C08998=1107.055,1.070,-52.195,179.860,6.489,149.225
C08999=1107.060,0.820,-52.181,179.860,6.484,149.224
C09000=1107.066,0.570,-52.166,179.859,6.479,149.223
C09001=1107.071,0.321,-52.151,179.859,6.476,149.223
C09002=1107.076,0.072,-52.137,179.858,6.471,149.222
C09003=1107.081,-0.178,-52.122,179.858,6.467,149.221
C09004=1107.086,-0.428,-52.108,179.857,6.462,149.220
C09005=1107.091,-0.678,-52.094,179.856,6.457,149.219
C09006=1107.096,-0.926,-52.079,179.855,6.453,149.218
C09007=1107.101,-1.176,-52.065,179.855,6.448,149.217
C09008=1107.106,-1.425,-52.051,179.854,6.444,149.217
C09009=1107.111,-1.675,-52.036,179.853,6.439,149.216
C09010=1107.116,-1.925,-52.022,179.853,6.434,149.215
C09011=1107.121,-2.175,-52.008,179.852,6.430,149.214
C09012=1107.126,-2.424,-51.994,179.851,6.425,149.213
C09013=1107.132,-2.673,-51.978,179.851,6.421,149.213
C09014=1107.136,-2.923,-51.964,179.851,6.417,149.212
C09015=1107.141,-3.172,-51.950,179.850,6.412,149.211
C09016=1107.146,-3.422,-51.935,179.849,6.408,149.210
C09017=1107.151,-3.636,-51.923,179.849,6.404,149.209
C09018=1107.155,-3.851,-51.911,179.848,6.400,149.209
C09019=1107.159,-4.065,-51.899,179.848,6.396,149.208
C09020=1107.164,-4.279,-51.887,179.848,6.392,149.207
C09021=1107.167,-4.493,-51.875,179.847,6.388,149.207
C09022=1107.172,-4.707,-51.863,179.846,6.384,149.206
C09023=1107.176,-4.921,-51.851,179.846,6.381,149.205
C09024=1107.181,-5.135,-51.838,179.845,6.376,149.204
C09025=1107.186,-5.385,-51.824,179.844,6.372,149.204
C09026=1107.191,-5.634,-51.810,179.844,6.367,149.203
C09027=1107.196,-5.884,-51.796,179.844,6.363,149.202
C09028=1107.201,-6.134,-51.781,179.843,6.359,149.201
C09029=1107.206,-6.383,-51.767,179.843,6.354,149.200
C09030=1107.211,-6.633,-51.753,179.842,6.349,149.199
C09031=1107.216,-6.882,-51.739,179.842,6.345,149.198
C09032=1107.221,-7.132,-51.725,179.841,6.340,149.198
C09033=1107.227,-7.381,-51.711,179.840,6.336,149.197
C09034=1107.232,-7.631,-51.696,179.839,6.331,149.196
C09035=1107.237,-7.881,-51.683,179.840,6.327,149.195
C09036=1107.241,-8.130,-51.669,179.839,6.323,149.194
C09037=1107.247,-8.379,-51.655,179.838,6.318,149.194
C09038=1107.252,-8.629,-51.641,179.838,6.313,149.193
C09039=1107.257,-8.879,-51.627,179.837,6.308,149.192
C09040=1107.262,-9.129,-51.612,179.836,6.304,149.191
C09041=1107.267,-9.378,-51.599,179.836,6.299,149.190
C09042=1107.272,-9.627,-51.584,179.835,6.295,149.189
C09043=1107.277,-9.878,-51.571,179.835,6.291,149.188
C09044=1107.282,-10.126,-51.557,179.834,6.286,149.188
C09045=1107.287,-10.376,-51.543,179.834,6.282,149.187
C09046=1107.292,-10.626,-51.529,179.833,6.277,149.186
C09047=1107.297,-10.875,-51.515,179.833,6.272,149.185
C09048=1107.303,-11.124,-51.501,179.832,6.268,149.184
C09049=1107.307,-11.374,-51.488,179.831,6.263,149.184
C09050=1107.312,-11.624,-51.473,179.831,6.259,149.183
C09051=1107.318,-11.873,-51.459,179.831,6.255,149.182
C09052=1107.323,-12.123,-51.445,179.830,6.250,149.181
C09053=1107.328,-12.373,-51.432,179.829,6.246,149.180
C09054=1107.333,-12.622,-51.418,179.829,6.241,149.179
C09055=1107.338,-12.872,-51.404,179.828,6.236,149.178
C09056=1107.343,-13.121,-51.390,179.828,6.231,149.177
C09057=1107.348,-13.371,-51.377,179.828,6.227,149.177
C09058=1107.353,-13.620,-51.363,179.827,6.223,149.176
C09059=1107.358,-13.870,-51.349,179.826,6.218,149.175
C09060=1107.363,-14.120,-51.335,179.826,6.214,149.174
C09061=1107.368,-14.369,-51.322,179.825,6.209,149.173
C09062=1107.373,-14.618,-51.308,179.825,6.204,149.172
C09063=1107.378,-14.868,-51.294,179.824,6.199,149.171
C09064=1107.383,-15.118,-51.280,179.825,6.196,149.170
C09065=1107.388,-15.367,-51.267,179.824,6.191,149.170
C09066=1107.393,-15.617,-51.253,179.823,6.186,149.169
C09067=1107.398,-15.867,-51.239,179.823,6.182,149.168
C09068=1107.404,-16.116,-51.226,179.822,6.177,149.167
C09069=1107.409,-16.366,-51.212,179.822,6.172,149.166
C09070=1107.414,-16.615,-51.198,179.821,6.168,149.165
C09071=1107.419,-16.865,-51.185,179.821,6.163,149.164
C09072=1107.424,-17.114,-51.171,179.821,6.159,149.164
C09073=1107.428,-17.329,-51.159,179.820,6.155,149.163
C09074=1107.433,-17.543,-51.147,179.819,6.151,149.162
C09075=1107.438,-17.758,-51.136,179.820,6.147,149.161
C09076=1107.441,-17.971,-51.125,179.819,6.143,149.161
C09077=1107.446,-18.185,-51.113,179.819,6.139,149.160
C09078=1107.450,-18.400,-51.101,179.818,6.135,149.159
C09079=1107.454,-18.614,-51.089,179.817,6.131,149.158
C09080=1107.459,-18.829,-51.078,179.817,6.127,149.157
C09081=1107.464,-19.078,-51.064,179.817,6.122,149.157
C09082=1107.469,-19.328,-51.051,179.816,6.118,149.156
C09083=1107.474,-19.577,-51.037,179.816,6.113,149.155
C09084=1107.479,-19.827,-51.024,179.816,6.109,149.154
C09085=1107.485,-20.077,-51.011,179.816,6.104,149.153
C09086=1107.489,-20.326,-50.997,179.815,6.100,149.152
C09087=1107.495,-20.576,-50.984,179.815,6.095,149.151
C09088=1107.499,-20.825,-50.970,179.814,6.090,149.150
C09089=1107.505,-21.075,-50.957,179.814,6.085,149.149
C09090=1107.510,-21.324,-50.943,179.813,6.081,149.148
C09091=1107.515,-21.574,-50.930,179.813,6.076,149.148
C09092=1107.520,-21.824,-50.917,179.813,6.072,149.147
C09093=1107.525,-22.073,-50.903,179.812,6.067,149.146
C09094=1107.531,-22.323,-50.890,179.812,6.062,149.145
C09095=1107.536,-22.572,-50.876,179.811,6.058,149.144
C09096=1107.541,-22.822,-50.863,179.811,6.053,149.143
C09097=1107.546,-23.071,-50.850,179.810,6.048,149.142
C09098=1107.551,-23.321,-50.836,179.810,6.044,149.141
C09099=1107.556,-23.570,-50.823,179.809,6.039,149.140
C09100=1107.561,-23.821,-50.810,179.809,6.034,149.139
C09101=1107.566,-24.069,-50.796,179.810,6.030,149.138
C09102=1107.571,-24.320,-50.783,179.809,6.025,149.137
C09103=1107.576,-24.569,-50.770,179.809,6.020,149.136
C09104=1107.581,-24.819,-50.757,179.808,6.016,149.136
C09105=1107.587,-25.068,-50.743,179.808,6.011,149.135
C09106=1107.591,-25.318,-50.730,179.807,6.006,149.134
C09107=1107.597,-25.568,-50.717,179.807,6.001,149.133
C09108=1107.602,-25.816,-50.704,179.807,5.996,149.132
C09109=1107.607,-26.067,-50.690,179.807,5.992,149.131
C09110=1107.612,-26.316,-50.678,179.807,5.987,149.130
C09111=1107.617,-26.566,-50.664,179.807,5.983,149.129
C09112=1107.622,-26.815,-50.651,179.807,5.979,149.128
C09113=1107.627,-27.065,-50.638,179.807,5.974,149.127
C09114=1107.633,-27.315,-50.625,179.807,5.970,149.126
C09115=1107.638,-27.564,-50.612,179.806,5.965,149.125
C09116=1107.642,-27.814,-50.599,179.806,5.961,149.124
C09117=1107.648,-28.063,-50.585,179.806,5.956,149.123
C09118=1107.652,-28.313,-50.572,179.807,5.952,149.122
C09119=1107.658,-28.563,-50.559,179.806,5.947,149.121
C09120=1107.663,-28.812,-50.546,179.806,5.943,149.120
C09121=1107.668,-29.062,-50.533,179.806,5.938,149.119
C09122=1107.674,-29.312,-50.520,179.805,5.934,149.118
C09123=1107.678,-29.561,-50.507,179.805,5.930,149.117
C09124=1107.683,-29.810,-50.494,179.805,5.925,149.117
C09125=1107.689,-30.060,-50.481,179.805,5.921,149.116
C09126=1107.693,-30.310,-50.468,179.805,5.916,149.115
C09127=1107.699,-30.559,-50.455,179.804,5.912,149.114
C09128=1107.704,-30.809,-50.442,179.804,5.908,149.113
C09129=1107.708,-31.023,-50.431,179.804,5.904,149.112
C09130=1107.713,-31.238,-50.420,179.804,5.900,149.111
C09131=1107.717,-31.452,-50.409,179.804,5.896,149.110
C09132=1107.722,-31.666,-50.397,179.803,5.892,149.110
C09133=1107.726,-31.880,-50.387,179.803,5.888,149.109
C09134=1107.730,-32.096,-50.375,179.803,5.884,149.108
C09135=1107.734,-32.310,-50.364,179.803,5.881,149.107
C09136=1107.739,-32.524,-50.353,179.802,5.877,149.107
C09137=1107.744,-32.774,-50.340,179.802,5.873,149.106
C09138=1107.750,-33.023,-50.327,179.802,5.868,149.105
C09139=1107.755,-33.273,-50.314,179.802,5.864,149.104
C09140=1107.759,-33.523,-50.301,179.801,5.859,149.103
C09141=1107.764,-33.772,-50.289,179.801,5.855,149.102
C09142=1107.770,-34.022,-50.276,179.801,5.851,149.101
C09143=1107.775,-34.272,-50.263,179.800,5.846,149.100
C09144=1107.780,-34.521,-50.250,179.800,5.842,149.100
C09145=1107.785,-34.770,-50.237,179.799,5.837,149.099
C09146=1107.790,-35.020,-50.225,179.799,5.833,149.098
C09147=1107.795,-35.270,-50.211,179.799,5.828,149.097
C09148=1107.801,-35.519,-50.199,179.798,5.823,149.096
C09149=1107.806,-35.768,-50.186,179.798,5.819,149.095
C09150=1107.810,-36.019,-50.173,179.797,5.814,149.094
C09151=1107.816,-36.268,-50.161,179.798,5.810,149.093
C09152=1107.822,-36.518,-50.148,179.797,5.806,149.093
C09153=1107.826,-36.768,-50.135,179.796,5.801,149.092
C09154=1107.831,-37.017,-50.122,179.796,5.796,149.091
C09155=1107.836,-37.267,-50.110,179.795,5.791,149.090
C09156=1107.841,-37.516,-50.097,179.795,5.787,149.089
C09157=1107.847,-37.766,-50.084,179.794,5.782,149.088
C09158=1107.852,-38.016,-50.071,179.795,5.778,149.087
C09159=1107.857,-38.266,-50.059,179.794,5.773,149.086
C09160=1107.862,-38.515,-50.047,179.794,5.769,149.085
C09161=1107.867,-38.764,-50.034,179.793,5.764,149.085
C09162=1107.872,-39.014,-50.021,179.793,5.759,149.084
C09163=1107.877,-39.264,-50.008,179.792,5.754,149.083
C09164=1107.883,-39.514,-49.997,179.792,5.750,149.082
C09165=1107.888,-39.763,-49.983,179.791,5.745,149.081
C09166=1107.894,-40.012,-49.971,179.791,5.740,149.080
C09167=1107.898,-40.263,-49.958,179.791,5.735,149.079
C09168=1107.904,-40.512,-49.946,179.790,5.731,149.078
C09169=1107.909,-40.762,-49.933,179.789,5.725,149.077
C09170=1107.914,-41.011,-49.921,179.789,5.720,149.076
C09171=1107.919,-41.260,-49.908,179.788,5.716,149.075
C09172=1107.924,-41.511,-49.896,179.788,5.710,149.074
C09173=1107.929,-41.760,-49.883,179.788,5.706,149.073
C09174=1107.934,-42.010,-49.871,179.787,5.701,149.072
C09175=1107.939,-42.260,-49.859,179.787,5.696,149.072
C09176=1107.945,-42.509,-49.846,179.786,5.691,149.071
C09177=1107.950,-42.758,-49.834,179.786,5.686,149.069
C09178=1107.955,-43.008,-49.822,179.786,5.681,149.069
C09179=1107.960,-43.258,-49.809,179.786,5.677,149.067
C09180=1107.965,-43.508,-49.796,179.786,5.671,149.066
C09181=1107.970,-43.757,-49.784,179.786,5.666,149.065
C09182=1107.975,-44.007,-49.772,179.786,5.662,149.064
C09183=1107.980,-44.256,-49.759,179.787,5.657,149.063
C09184=1107.986,-44.506,-49.747,179.787,5.653,149.062
C09185=1107.990,-44.720,-49.736,179.787,5.649,149.061
C09186=1107.995,-44.935,-49.725,179.787,5.644,149.060
C09187=1107.999,-45.150,-49.715,179.787,5.640,149.059
C09188=1108.003,-45.364,-49.704,179.787,5.636,149.058
C09189=1108.008,-45.578,-49.693,179.787,5.632,149.057
C09190=1108.013,-45.793,-49.683,179.788,5.628,149.056
C09191=1108.017,-46.007,-49.673,179.788,5.625,149.055
C09192=1108.021,-46.222,-49.663,179.788,5.621,149.055
C09193=1108.026,-46.471,-49.650,179.788,5.615,149.053
C09194=1108.031,-46.720,-49.638,179.788,5.610,149.052
C09195=1108.037,-46.970,-49.626,179.788,5.606,149.051
C09196=1108.041,-47.220,-49.613,179.788,5.601,149.050
C09197=1108.047,-47.470,-49.601,179.789,5.597,149.049
C09198=1108.052,-47.720,-49.588,179.789,5.592,149.048
C09199=1108.057,-47.970,-49.576,179.789,5.587,149.047
C09200=1108.062,-48.219,-49.564,179.789,5.583,149.046
C09201=1108.068,-48.469,-49.552,179.789,5.578,149.045
C09202=1108.072,-48.718,-49.540,179.789,5.573,149.044
C09203=1108.078,-48.968,-49.528,179.790,5.569,149.043
C09204=1108.083,-49.217,-49.515,179.790,5.563,149.041
C09205=1108.088,-49.467,-49.503,179.790,5.559,149.040
C09206=1108.094,-49.717,-49.492,179.790,5.554,149.039
C09207=1108.099,-49.966,-49.479,179.790,5.549,149.038
C09208=1108.104,-50.216,-49.467,179.791,5.545,149.037
C09209=1108.109,-50.465,-49.454,179.790,5.540,149.036
C09210=1108.114,-50.715,-49.443,179.790,5.535,149.035
C09211=1108.119,-50.964,-49.431,179.791,5.531,149.034
C09212=1108.125,-51.214,-49.419,179.791,5.526,149.033
C09213=1108.130,-51.464,-49.407,179.791,5.521,149.032
C09214=1108.135,-51.714,-49.394,179.791,5.517,149.031
C09215=1108.140,-51.964,-49.382,179.791,5.512,149.030
C09216=1108.145,-52.213,-49.370,179.792,5.507,149.029
C09217=1108.150,-52.462,-49.358,179.792,5.502,149.027
C09218=1108.155,-52.713,-49.346,179.791,5.498,149.026
C09219=1108.160,-52.962,-49.334,179.792,5.493,149.025
C09220=1108.166,-53.212,-49.322,179.792,5.488,149.024
C09221=1108.170,-53.462,-49.310,179.792,5.483,149.023
C09222=1108.176,-53.711,-49.298,179.792,5.479,149.022
C09223=1108.182,-53.961,-49.286,179.792,5.474,149.021
C09224=1108.187,-54.210,-49.274,179.792,5.469,149.020
C09225=1108.191,-54.459,-49.262,179.793,5.465,149.019
C09226=1108.197,-54.709,-49.251,179.793,5.460,149.018
C09227=1108.202,-54.959,-49.239,179.792,5.455,149.017
C09228=1108.208,-55.209,-49.227,179.793,5.451,149.016
C09229=1108.212,-55.458,-49.215,179.793,5.446,149.015
